(* PLC project batch, Dassault Systèmes ControlBuild 2020 *)
(* stored: creationDateTime 2019-04-23T11:14:51-01:00 *)

CONFIGURATION batch
  VAR_GLOBAL
    generalPanel/acknowledgePB AT 12 : BOOL := false;
    generalPanel/powerUp AT 6 : BOOL := false;
    generalPanel/emergencyStop AT 7 : BOOL := false;
    generalPanel/manualSwitch AT 8 : BOOL := false;
    generalPanel/autoSwitch AT 9 : BOOL := false;
    generalPanel/startCyclePB AT 10 : BOOL := false;
    generalPanel/endCyclePB AT 11 : BOOL := false;
    generalPanel/acknowledgePB/PB AT 12 : BOOL := false;
    generalPanel/acknowledgePB/action AT 26 : BOOL := false;
    generalPanel/acknowledgePB/timeCounter AT 17 : REAL := 0.0;
    generalPanel/acknowledgePB/pulseDuration AT 18 : REAL := 5.0;
    generalPanel/acknowledgePB/PBLogic AT 27 : BOOL := true;
    generalPanel/powerUp/PB AT 6 : BOOL := false;
    generalPanel/powerUp/action AT 28 : BOOL := false;
    generalPanel/powerUp/timeCounter AT 19 : REAL := 0.0;
    generalPanel/powerUp/pulseDuration AT 20 : REAL := 5.0;
    generalPanel/powerUp/PBLogic AT 29 : BOOL := true;
    generalPanel/modeSwitch/leftVariable AT 9 : BOOL := true;
    generalPanel/modeSwitch/rightVariable AT 8 : BOOL := false;
    generalPanel/modeSwitch/leftPosition AT 30 : BOOL := false;
    generalPanel/modeSwitch/rightPosition AT 31 : BOOL := false;
    generalPanel/startCyclePB/PB AT 10 : BOOL := false;
    generalPanel/startCyclePB/action AT 32 : BOOL := false;
    generalPanel/startCyclePB/timeCounter AT 21 : REAL := 0.0;
    generalPanel/startCyclePB/pulseDuration AT 22 : REAL := 5.0;
    generalPanel/startCyclePB/PBLogic AT 33 : BOOL := true;
    generalPanel/endCyclePB/PB AT 11 : BOOL := false;
    generalPanel/endCyclePB/action AT 34 : BOOL := false;
    generalPanel/endCyclePB/timeCounter AT 23 : REAL := 0.0;
    generalPanel/endCyclePB/pulseDuration AT 24 : REAL := 5.0;
    generalPanel/endCyclePB/PBLogic AT 35 : BOOL := true;
    generalPanel/bpCloture/PB AT 25 : BOOL := false;
    generalPanel/bpCloture/action AT 36 : BOOL := false;
    generalPanel/bpCloture/timeCounter AT 25 : REAL := 0.0;
    generalPanel/bpCloture/pulseDuration AT 26 : REAL := 5.0;
    generalPanel/bpCloture/PBLogic AT 37 : BOOL := true;
    generalPanel/emergencyStop/pb AT 7 : BOOL := false;
    generalPanel/emergencyStop/action AT 38 : BOOL := false;
    generalPanel/emergencyStop/PBLogic AT 39 : BOOL := false;
    recipe/flourWeight AT 523 : DINT := 0;
    recipe/syrup1Weight AT 524 : DINT := 0;
    recipe/syrup2Weight AT 525 : DINT := 0;
    recipe/syrup3Weight AT 526 : DINT := 0;
    recipe/recipeNumber AT 527 : DINT := 1;
    workingModes/powerUp AT 6 : BOOL := false;
    workingModes/emergencyStop AT 7 : BOOL := false;
    workingModes/manualSwitch AT 8 : BOOL := false;
    workingModes/autoSwitch AT 9 : BOOL := false;
    workingModes/startCyclePB AT 10 : BOOL := false;
    workingModes/endCyclePB AT 11 : BOOL := false;
    workingModes/acknowledgePB AT 12 : BOOL := false;
    workingModes/cycleEnd AT 13 : BOOL := false;
    workingModes/generalFault AT 14 : BOOL := false;
    workingModes/live AT 5 : BOOL := false;
    workingModes/autoMode AT 23 : BOOL := false;
    workingModes/manualMode AT 24 : BOOL := false;
    workingModes/cycleInProgress AT 15 : BOOL := false;
    workingModes/endCycleRequest AT 16 : BOOL := false;
    workingModes/emergencyStopState AT 40 : BOOL := false;
    management/cycleInProgress AT 15 : BOOL := false;
    management/endCycleRequest AT 16 : BOOL := false;
    management/kneadingOk AT 17 : BOOL := false;
    management/syrupWeighingOk AT 18 : BOOL := false;
    management/flourWeighingOk AT 19 : BOOL := false;
    management/cycleEnd AT 13 : BOOL := false;
    management/flourWeighingRq AT 20 : BOOL := false;
    management/syrupWeighingRq AT 21 : BOOL := false;
    management/kneadingRq AT 22 : BOOL := false;
    management/_X_10 AT 44 : BOOL := true;
    management/_X_11 AT 45 : BOOL := false;
    management/_X_12 AT 46 : BOOL := false;
    management/_X_13 AT 47 : BOOL := false;
    management/_X_14 AT 48 : BOOL := false;
    manufacturing/cycleInProgress AT 15 : BOOL := false;
    manufacturing/acknowledgePB AT 12 : BOOL := false;
    manufacturing/flourWeighingRequest AT 20 : BOOL := false;
    manufacturing/syrupWeighingRequest AT 21 : BOOL := false;
    manufacturing/kneadingRequest AT 22 : BOOL := false;
    manufacturing/autoMode AT 23 : BOOL := false;
    manufacturing/manualMode AT 24 : BOOL := false;
    manufacturing/flourWeight AT 523 : DINT := 0;
    manufacturing/syrup1Weight AT 524 : DINT := 0;
    manufacturing/syrup2Weight AT 525 : DINT := 0;
    manufacturing/syrup3Weight AT 526 : DINT := 0;
    manufacturing/generalFault AT 14 : BOOL := false;
    manufacturing/kneadingOK AT 17 : BOOL := false;
    manufacturing/flourWeighingOk AT 19 : BOOL := false;
    manufacturing/syrupWeighingOk AT 18 : BOOL := false;
    manufacturing/flour/cycleInProgress AT 15 : BOOL := false;
    manufacturing/flour/acknowledgePB AT 12 : BOOL := false;
    manufacturing/flour/weighingRequest AT 20 : BOOL := false;
    manufacturing/flour/flourWeight AT 523 : DINT := 0;
    manufacturing/flour/autoMode AT 23 : BOOL := false;
    manufacturing/flour/manualMode AT 24 : BOOL := false;
    manufacturing/flour/flourExtraction AT 28 : REAL := 0.0;
    manufacturing/flour/weighingOk AT 19 : BOOL := false;
    manufacturing/flour/fault AT 53 : BOOL := false;
    manufacturing/flour/airArrival/acknowledgePB AT 12 : BOOL := false;
    manufacturing/flour/airArrival/autoMode AT 23 : BOOL := false;
    manufacturing/flour/airArrival/manualMode AT 24 : BOOL := false;
    manufacturing/flour/airArrival/autoCloseCmd AT 62 : BOOL := false;
    manufacturing/flour/airArrival/autoOpenCmd AT 63 : BOOL := false;
    manufacturing/flour/airArrival/inputFlow AT 37 : REAL := 50.0;
    manufacturing/flour/airArrival/openedSensor AT 61 : BOOL := false;
    manufacturing/flour/airArrival/closedSensor AT 60 : BOOL := false;
    manufacturing/flour/airArrival/generalFault AT 66 : BOOL := false;
    manufacturing/flour/airArrival/outputFlow AT 39 : REAL := 0.0;
    manufacturing/flour/airArrival/percentOpening AT 36 : REAL := 0.0;
    manufacturing/flour/airArrival/panel1/closeValvePB AT 72 : BOOL := false;
    manufacturing/flour/airArrival/panel1/openValvePB AT 73 : BOOL := false;
    manufacturing/flour/airArrival/panel1/switch/leftVariable AT 72 : BOOL := false;
    manufacturing/flour/airArrival/panel1/switch/rightVariable AT 73 : BOOL := false;
    manufacturing/flour/airArrival/panel1/switch/leftPosition AT 76 : BOOL := false;
    manufacturing/flour/airArrival/panel1/switch/middlePosition AT 77 : BOOL := false;
    manufacturing/flour/airArrival/panel1/switch/rightPosition AT 78 : BOOL := false;
    manufacturing/flour/airArrival/cmdOfValve/autoMode AT 23 : BOOL := false;
    manufacturing/flour/airArrival/cmdOfValve/manualMode AT 24 : BOOL := false;
    manufacturing/flour/airArrival/cmdOfValve/closedSensorFB AT 60 : BOOL := false;
    manufacturing/flour/airArrival/cmdOfValve/openedSensorFB AT 61 : BOOL := false;
    manufacturing/flour/airArrival/cmdOfValve/autoCloseCmd AT 62 : BOOL := false;
    manufacturing/flour/airArrival/cmdOfValve/autoOpenCmd AT 63 : BOOL := false;
    manufacturing/flour/airArrival/cmdOfValve/closeValvePB AT 72 : BOOL := false;
    manufacturing/flour/airArrival/cmdOfValve/openValvePB AT 73 : BOOL := false;
    manufacturing/flour/airArrival/cmdOfValve/acknowledgePB AT 12 : BOOL := false;
    manufacturing/flour/airArrival/cmdOfValve/closeCmd AT 75 : BOOL := false;
    manufacturing/flour/airArrival/cmdOfValve/openCmd AT 74 : BOOL := false;
    manufacturing/flour/airArrival/cmdOfValve/generalFault AT 66 : BOOL := false;
    manufacturing/flour/airArrival/cmdOfValve/actions/autoMode AT 23 : BOOL := false;
    manufacturing/flour/airArrival/cmdOfValve/actions/manualMode AT 24 : BOOL := false;
    manufacturing/flour/airArrival/cmdOfValve/actions/autoCloseCmd AT 62 : BOOL := false;
    manufacturing/flour/airArrival/cmdOfValve/actions/autoOpenCmd AT 63 : BOOL := false;
    manufacturing/flour/airArrival/cmdOfValve/actions/closedSensorFB AT 60 : BOOL := false;
    manufacturing/flour/airArrival/cmdOfValve/actions/openedSensorFB AT 61 : BOOL := false;
    manufacturing/flour/airArrival/cmdOfValve/actions/closeValvePB AT 72 : BOOL := false;
    manufacturing/flour/airArrival/cmdOfValve/actions/openValvePB AT 73 : BOOL := false;
    manufacturing/flour/airArrival/cmdOfValve/actions/generalFault AT 66 : BOOL := false;
    manufacturing/flour/airArrival/cmdOfValve/actions/closeCmd AT 75 : BOOL := false;
    manufacturing/flour/airArrival/cmdOfValve/actions/openCmd AT 74 : BOOL := false;
    manufacturing/flour/airArrival/cmdOfValve/faults1/closeCmd AT 75 : BOOL := false;
    manufacturing/flour/airArrival/cmdOfValve/faults1/openCmd AT 74 : BOOL := false;
    manufacturing/flour/airArrival/cmdOfValve/faults1/closedSensorFB AT 60 : BOOL := false;
    manufacturing/flour/airArrival/cmdOfValve/faults1/openedSensorFB AT 61 : BOOL := false;
    manufacturing/flour/airArrival/cmdOfValve/faults1/acknowledgePB AT 12 : BOOL := false;
    manufacturing/flour/airArrival/cmdOfValve/faults1/generalFault AT 66 : BOOL := false;
    manufacturing/flour/airArrival/cmdOfValve/faults1/closedSensorFault AT 79 : BOOL := false;
    manufacturing/flour/airArrival/cmdOfValve/faults1/openedSensorFault AT 80 : BOOL := false;
    manufacturing/flour/airArrival/cmdOfValve/faults1/discordanceFault AT 81 : BOOL := false;
    manufacturing/flour/airArrival/cmdOfValve/faults1/presetMvt AT 542 : TIME := T#0h0m4s0ms;
    manufacturing/flour/airArrival/cmdOfValve/faults1/presetDiscordance AT 546 : TIME := T#0h0m0s200ms;
    manufacturing/flour/airArrival/valve/voltage380 AT 71 : BOOL := true;
    manufacturing/flour/airArrival/valve/cmdSupply AT 70 : BOOL := true;
    manufacturing/flour/airArrival/valve/sensorSupply AT 69 : BOOL := true;
    manufacturing/flour/airArrival/valve/openCmd AT 74 : BOOL := false;
    manufacturing/flour/airArrival/valve/closeCmd AT 75 : BOOL := false;
    manufacturing/flour/airArrival/valve/inputFlow AT 37 : REAL := 50.0;
    manufacturing/flour/airArrival/valve/openedSensor AT 61 : BOOL := false;
    manufacturing/flour/airArrival/valve/closedSensor AT 60 : BOOL := false;
    manufacturing/flour/airArrival/valve/outputFlow AT 39 : REAL := 0.0;
    manufacturing/flour/airArrival/valve/percentOpening AT 36 : REAL := 0.0;
    manufacturing/flour/airArrival/valve/increment AT 45 : REAL := 0.0;
    manufacturing/flour/airArrival/valve/memoOpen AT 91 : BOOL := false;
    manufacturing/flour/airArrival/valve/memoClose AT 92 : BOOL := false;
    manufacturing/flour/airArrival/valve/openState AT 93 : BOOL := false;
    manufacturing/flour/airArrival/valve/closeState AT 94 : BOOL := false;
    manufacturing/flour/airArrival/valve/openingVal AT 46 : REAL := 0.0;
    manufacturing/flour/airArrival/valve/unit AT 47 : REAL := 0.0;
    manufacturing/flour/airArrival/valve/openingTime AT 48 : REAL := 0.5;
    manufacturing/flour/airArrival/valve/openedSensorLogic AT 95 : BOOL := true;
    manufacturing/flour/airArrival/valve/closedSensorLogic AT 96 : BOOL := true;
    manufacturing/flour/airArrival/valve/flowMax AT 49 : REAL := 10000.0;
    manufacturing/flour/airArrival/valve/flowPerHour AT 97 : BOOL := true;
    manufacturing/flour/airArrival/valve/flowPerMinute AT 98 : BOOL := false;
    manufacturing/flour/airArrival/valve/d_locking AT 99 : BOOL := false;
    manufacturing/flour/airArrival/valve/v_d_locking AT 50 : REAL := 2.0;
    manufacturing/flour/airArrival/valve/d_flow AT 100 : BOOL := false;
    manufacturing/flour/airArrival/valve/v_d_flow AT 51 : REAL := 2.0;
    manufacturing/flour/airArrival/valve/d_electrical AT 101 : BOOL := false;
    manufacturing/flour/airArrival/valve/v_d_electrical AT 102 : BOOL := false;
    manufacturing/flour/airArrival/valve/d_closedSensor AT 103 : BOOL := false;
    manufacturing/flour/airArrival/valve/v_d_closedSensor AT 104 : BOOL := false;
    manufacturing/flour/airArrival/valve/d_openedSensor AT 105 : BOOL := false;
    manufacturing/flour/airArrival/valve/v_d_openedSensor AT 106 : BOOL := false;
    manufacturing/flour/extractingValve/acknowledgePB AT 12 : BOOL := false;
    manufacturing/flour/extractingValve/autoMode AT 23 : BOOL := false;
    manufacturing/flour/extractingValve/manualMode AT 24 : BOOL := false;
    manufacturing/flour/extractingValve/autoCloseCmd AT 64 : BOOL := false;
    manufacturing/flour/extractingValve/autoOpenCmd AT 65 : BOOL := false;
    manufacturing/flour/extractingValve/inputFlow AT 38 : REAL := 0.0;
    manufacturing/flour/extractingValve/openedSensor AT 59 : BOOL := false;
    manufacturing/flour/extractingValve/closedSensor AT 58 : BOOL := false;
    manufacturing/flour/extractingValve/generalFault AT 68 : BOOL := false;
    manufacturing/flour/extractingValve/outputFlow AT 28 : REAL := 0.0;
    manufacturing/flour/extractingValve/percentOpening AT 35 : REAL := 0.0;
    manufacturing/flour/extractingValve/panel1/closeValvePB AT 110 : BOOL := false;
    manufacturing/flour/extractingValve/panel1/openValvePB AT 111 : BOOL := false;
    manufacturing/flour/extractingValve/panel1/switch/leftVariable AT 110 : BOOL := false;
    manufacturing/flour/extractingValve/panel1/switch/rightVariable AT 111 : BOOL := false;
    manufacturing/flour/extractingValve/panel1/switch/leftPosition AT 114 : BOOL := false;
    manufacturing/flour/extractingValve/panel1/switch/middlePosition AT 115 : BOOL := false;
    manufacturing/flour/extractingValve/panel1/switch/rightPosition AT 116 : BOOL := false;
    manufacturing/flour/extractingValve/cmdOfValve/autoMode AT 23 : BOOL := false;
    manufacturing/flour/extractingValve/cmdOfValve/manualMode AT 24 : BOOL := false;
    manufacturing/flour/extractingValve/cmdOfValve/closedSensorFB AT 58 : BOOL := false;
    manufacturing/flour/extractingValve/cmdOfValve/openedSensorFB AT 59 : BOOL := false;
    manufacturing/flour/extractingValve/cmdOfValve/autoCloseCmd AT 64 : BOOL := false;
    manufacturing/flour/extractingValve/cmdOfValve/autoOpenCmd AT 65 : BOOL := false;
    manufacturing/flour/extractingValve/cmdOfValve/closeValvePB AT 110 : BOOL := false;
    manufacturing/flour/extractingValve/cmdOfValve/openValvePB AT 111 : BOOL := false;
    manufacturing/flour/extractingValve/cmdOfValve/acknowledgePB AT 12 : BOOL := false;
    manufacturing/flour/extractingValve/cmdOfValve/closeCmd AT 113 : BOOL := false;
    manufacturing/flour/extractingValve/cmdOfValve/openCmd AT 112 : BOOL := false;
    manufacturing/flour/extractingValve/cmdOfValve/generalFault AT 68 : BOOL := false;
    manufacturing/flour/extractingValve/cmdOfValve/actions/autoMode AT 23 : BOOL := false;
    manufacturing/flour/extractingValve/cmdOfValve/actions/manualMode AT 24 : BOOL := false;
    manufacturing/flour/extractingValve/cmdOfValve/actions/autoCloseCmd AT 64 : BOOL := false;
    manufacturing/flour/extractingValve/cmdOfValve/actions/autoOpenCmd AT 65 : BOOL := false;
    manufacturing/flour/extractingValve/cmdOfValve/actions/closedSensorFB AT 58 : BOOL := false;
    manufacturing/flour/extractingValve/cmdOfValve/actions/openedSensorFB AT 59 : BOOL := false;
    manufacturing/flour/extractingValve/cmdOfValve/actions/closeValvePB AT 110 : BOOL := false;
    manufacturing/flour/extractingValve/cmdOfValve/actions/openValvePB AT 111 : BOOL := false;
    manufacturing/flour/extractingValve/cmdOfValve/actions/generalFault AT 68 : BOOL := false;
    manufacturing/flour/extractingValve/cmdOfValve/actions/closeCmd AT 113 : BOOL := false;
    manufacturing/flour/extractingValve/cmdOfValve/actions/openCmd AT 112 : BOOL := false;
    manufacturing/flour/extractingValve/cmdOfValve/faults1/closeCmd AT 113 : BOOL := false;
    manufacturing/flour/extractingValve/cmdOfValve/faults1/openCmd AT 112 : BOOL := false;
    manufacturing/flour/extractingValve/cmdOfValve/faults1/closedSensorFB AT 58 : BOOL := false;
    manufacturing/flour/extractingValve/cmdOfValve/faults1/openedSensorFB AT 59 : BOOL := false;
    manufacturing/flour/extractingValve/cmdOfValve/faults1/acknowledgePB AT 12 : BOOL := false;
    manufacturing/flour/extractingValve/cmdOfValve/faults1/generalFault AT 68 : BOOL := false;
    manufacturing/flour/extractingValve/cmdOfValve/faults1/closedSensorFault AT 117 : BOOL := false;
    manufacturing/flour/extractingValve/cmdOfValve/faults1/openedSensorFault AT 118 : BOOL := false;
    manufacturing/flour/extractingValve/cmdOfValve/faults1/discordanceFault AT 119 : BOOL := false;
    manufacturing/flour/extractingValve/cmdOfValve/faults1/presetMvt AT 583 : TIME := T#0h0m4s0ms;
    manufacturing/flour/extractingValve/cmdOfValve/faults1/presetDiscordance AT 587 : TIME := T#0h0m0s200ms;
    manufacturing/flour/extractingValve/valve/voltage380 AT 109 : BOOL := true;
    manufacturing/flour/extractingValve/valve/cmdSupply AT 108 : BOOL := true;
    manufacturing/flour/extractingValve/valve/sensorSupply AT 107 : BOOL := true;
    manufacturing/flour/extractingValve/valve/openCmd AT 112 : BOOL := false;
    manufacturing/flour/extractingValve/valve/closeCmd AT 113 : BOOL := false;
    manufacturing/flour/extractingValve/valve/inputFlow AT 38 : REAL := 0.0;
    manufacturing/flour/extractingValve/valve/openedSensor AT 59 : BOOL := false;
    manufacturing/flour/extractingValve/valve/closedSensor AT 58 : BOOL := false;
    manufacturing/flour/extractingValve/valve/outputFlow AT 28 : REAL := 0.0;
    manufacturing/flour/extractingValve/valve/percentOpening AT 35 : REAL := 0.0;
    manufacturing/flour/extractingValve/valve/increment AT 55 : REAL := 0.0;
    manufacturing/flour/extractingValve/valve/memoOpen AT 129 : BOOL := false;
    manufacturing/flour/extractingValve/valve/memoClose AT 130 : BOOL := false;
    manufacturing/flour/extractingValve/valve/openState AT 131 : BOOL := false;
    manufacturing/flour/extractingValve/valve/closeState AT 132 : BOOL := false;
    manufacturing/flour/extractingValve/valve/openingVal AT 56 : REAL := 0.0;
    manufacturing/flour/extractingValve/valve/unit AT 57 : REAL := 0.0;
    manufacturing/flour/extractingValve/valve/openingTime AT 58 : REAL := 0.5;
    manufacturing/flour/extractingValve/valve/openedSensorLogic AT 133 : BOOL := true;
    manufacturing/flour/extractingValve/valve/closedSensorLogic AT 134 : BOOL := true;
    manufacturing/flour/extractingValve/valve/flowMax AT 59 : REAL := 10000.0;
    manufacturing/flour/extractingValve/valve/flowPerHour AT 135 : BOOL := true;
    manufacturing/flour/extractingValve/valve/flowPerMinute AT 136 : BOOL := false;
    manufacturing/flour/extractingValve/valve/d_locking AT 137 : BOOL := false;
    manufacturing/flour/extractingValve/valve/v_d_locking AT 60 : REAL := 2.0;
    manufacturing/flour/extractingValve/valve/d_flow AT 138 : BOOL := false;
    manufacturing/flour/extractingValve/valve/v_d_flow AT 61 : REAL := 2.0;
    manufacturing/flour/extractingValve/valve/d_electrical AT 139 : BOOL := false;
    manufacturing/flour/extractingValve/valve/v_d_electrical AT 140 : BOOL := false;
    manufacturing/flour/extractingValve/valve/d_closedSensor AT 141 : BOOL := false;
    manufacturing/flour/extractingValve/valve/v_d_closedSensor AT 142 : BOOL := false;
    manufacturing/flour/extractingValve/valve/d_openedSensor AT 143 : BOOL := false;
    manufacturing/flour/extractingValve/valve/v_d_openedSensor AT 144 : BOOL := false;
    manufacturing/flour/airExtraction/acknowledgePB AT 12 : BOOL := false;
    manufacturing/flour/airExtraction/autoMode AT 23 : BOOL := false;
    manufacturing/flour/airExtraction/manualMode AT 24 : BOOL := false;
    manufacturing/flour/airExtraction/autoCloseCmd AT 64 : BOOL := false;
    manufacturing/flour/airExtraction/autoOpenCmd AT 65 : BOOL := false;
    manufacturing/flour/airExtraction/inputFlow AT 34 : REAL := 0.0;
    manufacturing/flour/airExtraction/openedSensor AT 57 : BOOL := false;
    manufacturing/flour/airExtraction/closedSensor AT 56 : BOOL := false;
    manufacturing/flour/airExtraction/generalFault AT 67 : BOOL := false;
    manufacturing/flour/airExtraction/outputFlow AT 33 : REAL := 0.0;
    manufacturing/flour/airExtraction/percentOpening AT 32 : REAL := 0.0;
    manufacturing/flour/airExtraction/panel1/closeValvePB AT 148 : BOOL := false;
    manufacturing/flour/airExtraction/panel1/openValvePB AT 149 : BOOL := false;
    manufacturing/flour/airExtraction/panel1/switch/leftVariable AT 148 : BOOL := false;
    manufacturing/flour/airExtraction/panel1/switch/rightVariable AT 149 : BOOL := false;
    manufacturing/flour/airExtraction/panel1/switch/leftPosition AT 152 : BOOL := false;
    manufacturing/flour/airExtraction/panel1/switch/middlePosition AT 153 : BOOL := false;
    manufacturing/flour/airExtraction/panel1/switch/rightPosition AT 154 : BOOL := false;
    manufacturing/flour/airExtraction/cmdOfValve/autoMode AT 23 : BOOL := false;
    manufacturing/flour/airExtraction/cmdOfValve/manualMode AT 24 : BOOL := false;
    manufacturing/flour/airExtraction/cmdOfValve/closedSensorFB AT 56 : BOOL := false;
    manufacturing/flour/airExtraction/cmdOfValve/openedSensorFB AT 57 : BOOL := false;
    manufacturing/flour/airExtraction/cmdOfValve/autoCloseCmd AT 64 : BOOL := false;
    manufacturing/flour/airExtraction/cmdOfValve/autoOpenCmd AT 65 : BOOL := false;
    manufacturing/flour/airExtraction/cmdOfValve/closeValvePB AT 148 : BOOL := false;
    manufacturing/flour/airExtraction/cmdOfValve/openValvePB AT 149 : BOOL := false;
    manufacturing/flour/airExtraction/cmdOfValve/acknowledgePB AT 12 : BOOL := false;
    manufacturing/flour/airExtraction/cmdOfValve/closeCmd AT 151 : BOOL := false;
    manufacturing/flour/airExtraction/cmdOfValve/openCmd AT 150 : BOOL := false;
    manufacturing/flour/airExtraction/cmdOfValve/generalFault AT 67 : BOOL := false;
    manufacturing/flour/airExtraction/cmdOfValve/actions/autoMode AT 23 : BOOL := false;
    manufacturing/flour/airExtraction/cmdOfValve/actions/manualMode AT 24 : BOOL := false;
    manufacturing/flour/airExtraction/cmdOfValve/actions/autoCloseCmd AT 64 : BOOL := false;
    manufacturing/flour/airExtraction/cmdOfValve/actions/autoOpenCmd AT 65 : BOOL := false;
    manufacturing/flour/airExtraction/cmdOfValve/actions/closedSensorFB AT 56 : BOOL := false;
    manufacturing/flour/airExtraction/cmdOfValve/actions/openedSensorFB AT 57 : BOOL := false;
    manufacturing/flour/airExtraction/cmdOfValve/actions/closeValvePB AT 148 : BOOL := false;
    manufacturing/flour/airExtraction/cmdOfValve/actions/openValvePB AT 149 : BOOL := false;
    manufacturing/flour/airExtraction/cmdOfValve/actions/generalFault AT 67 : BOOL := false;
    manufacturing/flour/airExtraction/cmdOfValve/actions/closeCmd AT 151 : BOOL := false;
    manufacturing/flour/airExtraction/cmdOfValve/actions/openCmd AT 150 : BOOL := false;
    manufacturing/flour/airExtraction/cmdOfValve/faults1/closeCmd AT 151 : BOOL := false;
    manufacturing/flour/airExtraction/cmdOfValve/faults1/openCmd AT 150 : BOOL := false;
    manufacturing/flour/airExtraction/cmdOfValve/faults1/closedSensorFB AT 56 : BOOL := false;
    manufacturing/flour/airExtraction/cmdOfValve/faults1/openedSensorFB AT 57 : BOOL := false;
    manufacturing/flour/airExtraction/cmdOfValve/faults1/acknowledgePB AT 12 : BOOL := false;
    manufacturing/flour/airExtraction/cmdOfValve/faults1/generalFault AT 67 : BOOL := false;
    manufacturing/flour/airExtraction/cmdOfValve/faults1/closedSensorFault AT 155 : BOOL := false;
    manufacturing/flour/airExtraction/cmdOfValve/faults1/openedSensorFault AT 156 : BOOL := false;
    manufacturing/flour/airExtraction/cmdOfValve/faults1/discordanceFault AT 157 : BOOL := false;
    manufacturing/flour/airExtraction/cmdOfValve/faults1/presetMvt AT 624 : TIME := T#0h0m4s0ms;
    manufacturing/flour/airExtraction/cmdOfValve/faults1/presetDiscordance AT 628 : TIME := T#0h0m0s200ms;
    manufacturing/flour/airExtraction/valve/voltage380 AT 147 : BOOL := true;
    manufacturing/flour/airExtraction/valve/cmdSupply AT 146 : BOOL := true;
    manufacturing/flour/airExtraction/valve/sensorSupply AT 145 : BOOL := true;
    manufacturing/flour/airExtraction/valve/openCmd AT 150 : BOOL := false;
    manufacturing/flour/airExtraction/valve/closeCmd AT 151 : BOOL := false;
    manufacturing/flour/airExtraction/valve/inputFlow AT 34 : REAL := 0.0;
    manufacturing/flour/airExtraction/valve/openedSensor AT 57 : BOOL := false;
    manufacturing/flour/airExtraction/valve/closedSensor AT 56 : BOOL := false;
    manufacturing/flour/airExtraction/valve/outputFlow AT 33 : REAL := 0.0;
    manufacturing/flour/airExtraction/valve/percentOpening AT 32 : REAL := 0.0;
    manufacturing/flour/airExtraction/valve/increment AT 65 : REAL := 0.0;
    manufacturing/flour/airExtraction/valve/memoOpen AT 167 : BOOL := false;
    manufacturing/flour/airExtraction/valve/memoClose AT 168 : BOOL := false;
    manufacturing/flour/airExtraction/valve/openState AT 169 : BOOL := false;
    manufacturing/flour/airExtraction/valve/closeState AT 170 : BOOL := false;
    manufacturing/flour/airExtraction/valve/openingVal AT 66 : REAL := 0.0;
    manufacturing/flour/airExtraction/valve/unit AT 67 : REAL := 0.0;
    manufacturing/flour/airExtraction/valve/openingTime AT 68 : REAL := 0.5;
    manufacturing/flour/airExtraction/valve/openedSensorLogic AT 171 : BOOL := true;
    manufacturing/flour/airExtraction/valve/closedSensorLogic AT 172 : BOOL := true;
    manufacturing/flour/airExtraction/valve/flowMax AT 69 : REAL := 10000.0;
    manufacturing/flour/airExtraction/valve/flowPerHour AT 173 : BOOL := true;
    manufacturing/flour/airExtraction/valve/flowPerMinute AT 174 : BOOL := false;
    manufacturing/flour/airExtraction/valve/d_locking AT 175 : BOOL := false;
    manufacturing/flour/airExtraction/valve/v_d_locking AT 70 : REAL := 2.0;
    manufacturing/flour/airExtraction/valve/d_flow AT 176 : BOOL := false;
    manufacturing/flour/airExtraction/valve/v_d_flow AT 71 : REAL := 2.0;
    manufacturing/flour/airExtraction/valve/d_electrical AT 177 : BOOL := false;
    manufacturing/flour/airExtraction/valve/v_d_electrical AT 178 : BOOL := false;
    manufacturing/flour/airExtraction/valve/d_closedSensor AT 179 : BOOL := false;
    manufacturing/flour/airExtraction/valve/v_d_closedSensor AT 180 : BOOL := false;
    manufacturing/flour/airExtraction/valve/d_openedSensor AT 181 : BOOL := false;
    manufacturing/flour/airExtraction/valve/v_d_openedSensor AT 182 : BOOL := false;
    manufacturing/flour/flourWeighing/inletFlow AT 39 : REAL := 0.0;
    manufacturing/flour/flourWeighing/outletFlow AT 28 : REAL := 0.0;
    manufacturing/flour/flourWeighing/tankLevel AT 40 : REAL := 0.0;
    manufacturing/flour/flourWeighing/percent AT 72 : REAL := 0.0;
    manufacturing/flour/flourWeighing/capacity AT 73 : REAL := 100.0;
    manufacturing/flour/flourWeighing/d_level AT 183 : BOOL := false;
    manufacturing/flour/flourWeighing/v_d_level AT 74 : REAL := 0.0;
    manufacturing/flour/flow/inputFlow AT 40 : REAL := 0.0;
    manufacturing/flour/flow/outputFlow AT 38 : REAL := 0.0;
    manufacturing/flour/flow/unit AT 75 : REAL := 0.0;
    manufacturing/flour/flow/flowMax AT 76 : REAL := 20000.0;
    manufacturing/flour/flow/flowPerHour AT 184 : BOOL := true;
    manufacturing/flour/flow/flowPerMinute AT 185 : BOOL := false;
    manufacturing/flour/level/measure AT 40 : REAL := 0.0;
    manufacturing/flour/level/sensorSupply AT 55 : BOOL := true;
    manufacturing/flour/level/realValue AT 41 : REAL := 0.0;
    manufacturing/flour/level/intValue AT 31 : REAL := 0.0;
    manufacturing/flour/level/dintValue AT 30 : REAL := 0.0;
    manufacturing/flour/level/tmp AT 656 : DINT := 0;
    manufacturing/flour/level/localValue AT 77 : REAL := 0.0;
    manufacturing/flour/level/nbDigit AT 657 : SINT := 2;
    manufacturing/flour/level/d_value AT 186 : BOOL := false;
    manufacturing/flour/level/v_d_value AT 78 : REAL := 0.0;
    manufacturing/flour/faults1/generalFault3 AT 66 : BOOL := false;
    manufacturing/flour/faults1/generalFault2 AT 67 : BOOL := false;
    manufacturing/flour/faults1/generalFault1 AT 68 : BOOL := false;
    manufacturing/flour/faults1/fault AT 53 : BOOL := false;
    manufacturing/flour/flourManagement/weighingRequest AT 20 : BOOL := false;
    manufacturing/flour/flourManagement/cycleInProgress AT 15 : BOOL := false;
    manufacturing/flour/flourManagement/weighedWeight AT 532 : DINT := 0;
    manufacturing/flour/flourManagement/flourWeight AT 523 : DINT := 0;
    manufacturing/flour/flourManagement/weighingOk AT 19 : BOOL := false;
    manufacturing/flour/flourManagement/introduceFlour AT 63 : BOOL := false;
    manufacturing/flour/flourManagement/introFlourEnd AT 62 : BOOL := false;
    manufacturing/flour/flourManagement/exitFlour AT 65 : BOOL := false;
    manufacturing/flour/flourManagement/exitFlourEnd AT 64 : BOOL := false;
    manufacturing/flour/flourManagement/totalWeight AT 658 : DINT := 0;
    manufacturing/flour/flourManagement/endOfWeighing AT 187 : BOOL := false;
    manufacturing/flour/flourManagement/_X_10 AT 188 : BOOL := true;
    manufacturing/flour/flourManagement/_X_11 AT 189 : BOOL := false;
    manufacturing/flour/flourManagement/_X_12 AT 190 : BOOL := false;
    manufacturing/flour/flourManagement/_X_13 AT 191 : BOOL := false;
    manufacturing/flour/flourManagement/_X_14 AT 192 : BOOL := false;
    manufacturing/flour/flourManagement/_X_15 AT 193 : BOOL := false;
    manufacturing/flour/flourManagement/maxWeight AT 659 : DINT := 100;
    manufacturing/flour/scale/inputValue AT 41 : REAL := 0.0;
    manufacturing/flour/scale/realValue AT 29 : REAL := 0.0;
    manufacturing/flour/scale/dintValue AT 532 : DINT := 0;
    manufacturing/flour/scale/intValue AT 531 : INT := 0;
    manufacturing/flour/scale/a AT 79 : REAL := 0.0;
    manufacturing/flour/scale/b AT 80 : REAL := 0.0;
    manufacturing/flour/scale/k AT 81 : REAL := 0.0;
    manufacturing/flour/scale/minInput AT 82 : REAL := 0.0;
    manufacturing/flour/scale/maxInput AT 83 : REAL := 100.0;
    manufacturing/flour/scale/minOutput AT 84 : REAL := 0.0;
    manufacturing/flour/scale/maxOutput AT 85 : REAL := 100.0;
    manufacturing/flour/scale/d_scale AT 198 : BOOL := false;
    manufacturing/flour/scale/v_d_scale AT 86 : REAL := 0.0;
    manufacturing/syrup/syrup1Weight AT 524 : DINT := 0;
    manufacturing/syrup/syrup2Weight AT 525 : DINT := 0;
    manufacturing/syrup/syrup3Weight AT 526 : DINT := 0;
    manufacturing/syrup/cycleInProgress AT 15 : BOOL := false;
    manufacturing/syrup/weighingRequest AT 21 : BOOL := false;
    manufacturing/syrup/acknowledgePB AT 12 : BOOL := false;
    manufacturing/syrup/autoMode AT 23 : BOOL := false;
    manufacturing/syrup/manualMode AT 24 : BOOL := false;
    manufacturing/syrup/weighingOk AT 18 : BOOL := false;
    manufacturing/syrup/fault AT 54 : BOOL := false;
    manufacturing/syrup/syrupExtraction AT 27 : REAL := 0.0;
    manufacturing/syrup/flow/inputFlow AT 97 : REAL := 0.0;
    manufacturing/syrup/flow/outputFlow AT 98 : REAL := 0.0;
    manufacturing/syrup/flow/unit AT 104 : REAL := 0.0;
    manufacturing/syrup/flow/flowMax AT 105 : REAL := 40000.0;
    manufacturing/syrup/flow/flowPerHour AT 220 : BOOL := true;
    manufacturing/syrup/flow/flowPerMinute AT 221 : BOOL := false;
    manufacturing/syrup/syrupManagement/weighingRequest AT 21 : BOOL := false;
    manufacturing/syrup/syrupManagement/cycleInProgress AT 15 : BOOL := false;
    manufacturing/syrup/syrupManagement/weighingWeight AT 662 : DINT := 0;
    manufacturing/syrup/syrupManagement/syrup1Weight AT 524 : DINT := 0;
    manufacturing/syrup/syrupManagement/syrup2Weight AT 525 : DINT := 0;
    manufacturing/syrup/syrupManagement/syrup3Weight AT 526 : DINT := 0;
    manufacturing/syrup/syrupManagement/weighingOk AT 18 : BOOL := false;
    manufacturing/syrup/syrupManagement/introduceS1 AT 209 : BOOL := false;
    manufacturing/syrup/syrupManagement/introS1End AT 208 : BOOL := false;
    manufacturing/syrup/syrupManagement/introduceS2 AT 211 : BOOL := false;
    manufacturing/syrup/syrupManagement/introS2End AT 210 : BOOL := false;
    manufacturing/syrup/syrupManagement/introduceS3 AT 213 : BOOL := false;
    manufacturing/syrup/syrupManagement/introS3End AT 212 : BOOL := false;
    manufacturing/syrup/syrupManagement/exitSyrup AT 215 : BOOL := false;
    manufacturing/syrup/syrupManagement/exitSyrupEnd AT 214 : BOOL := false;
    manufacturing/syrup/syrupManagement/totalWeight AT 663 : DINT := 0;
    manufacturing/syrup/syrupManagement/weighingS1 AT 222 : BOOL := false;
    manufacturing/syrup/syrupManagement/weighingS2 AT 223 : BOOL := false;
    manufacturing/syrup/syrupManagement/weighingS3 AT 224 : BOOL := false;
    manufacturing/syrup/syrupManagement/weighingS1Ok AT 225 : BOOL := false;
    manufacturing/syrup/syrupManagement/weighingS2Ok AT 226 : BOOL := false;
    manufacturing/syrup/syrupManagement/weighingS3Ok AT 227 : BOOL := false;
    manufacturing/syrup/syrupManagement/endOfWeighingS3 AT 228 : BOOL := false;
    manufacturing/syrup/syrupManagement/endOfWeighingS2 AT 229 : BOOL := false;
    manufacturing/syrup/syrupManagement/endOfWeighingS1 AT 230 : BOOL := false;
    manufacturing/syrup/syrupManagement/_X_10 AT 231 : BOOL := true;
    manufacturing/syrup/syrupManagement/_X_11 AT 232 : BOOL := false;
    manufacturing/syrup/syrupManagement/_X_12 AT 233 : BOOL := false;
    manufacturing/syrup/syrupManagement/_X_13 AT 234 : BOOL := false;
    manufacturing/syrup/syrupManagement/_X_14 AT 235 : BOOL := false;
    manufacturing/syrup/syrupManagement/_X_15 AT 236 : BOOL := false;
    manufacturing/syrup/syrupManagement/_X_20 AT 237 : BOOL := true;
    manufacturing/syrup/syrupManagement/_X_21 AT 238 : BOOL := false;
    manufacturing/syrup/syrupManagement/_X_22 AT 239 : BOOL := false;
    manufacturing/syrup/syrupManagement/_X_23 AT 240 : BOOL := false;
    manufacturing/syrup/syrupManagement/_X_24 AT 241 : BOOL := false;
    manufacturing/syrup/syrupManagement/_X_30 AT 242 : BOOL := true;
    manufacturing/syrup/syrupManagement/_X_31 AT 243 : BOOL := false;
    manufacturing/syrup/syrupManagement/_X_32 AT 244 : BOOL := false;
    manufacturing/syrup/syrupManagement/_X_33 AT 247 : BOOL := false;
    manufacturing/syrup/syrupManagement/_X_34 AT 245 : BOOL := false;
    manufacturing/syrup/syrupManagement/_X_35 AT 246 : BOOL := false;
    manufacturing/syrup/syrupManagement/_X_40 AT 248 : BOOL := true;
    manufacturing/syrup/syrupManagement/_X_41 AT 249 : BOOL := false;
    manufacturing/syrup/syrupManagement/_X_42 AT 250 : BOOL := false;
    manufacturing/syrup/syrupManagement/_X_43 AT 253 : BOOL := false;
    manufacturing/syrup/syrupManagement/_X_44 AT 251 : BOOL := false;
    manufacturing/syrup/syrupManagement/_X_45 AT 252 : BOOL := false;
    manufacturing/syrup/syrupManagement/maxWeight AT 664 : DINT := 200;
    manufacturing/syrup/arrivalValveSyrup1/acknowledgePB AT 12 : BOOL := false;
    manufacturing/syrup/arrivalValveSyrup1/autoMode AT 23 : BOOL := false;
    manufacturing/syrup/arrivalValveSyrup1/manualMode AT 24 : BOOL := false;
    manufacturing/syrup/arrivalValveSyrup1/autoCloseCmd AT 208 : BOOL := false;
    manufacturing/syrup/arrivalValveSyrup1/autoOpenCmd AT 209 : BOOL := false;
    manufacturing/syrup/arrivalValveSyrup1/inputFlow AT 96 : REAL := 50.0;
    manufacturing/syrup/arrivalValveSyrup1/openedSensor AT 207 : BOOL := false;
    manufacturing/syrup/arrivalValveSyrup1/closedSensor AT 206 : BOOL := false;
    manufacturing/syrup/arrivalValveSyrup1/generalFault AT 216 : BOOL := false;
    manufacturing/syrup/arrivalValveSyrup1/outputFlow AT 99 : REAL := 0.0;
    manufacturing/syrup/arrivalValveSyrup1/percentOpening AT 95 : REAL := 0.0;
    manufacturing/syrup/arrivalValveSyrup1/panel1/closeValvePB AT 273 : BOOL := false;
    manufacturing/syrup/arrivalValveSyrup1/panel1/openValvePB AT 274 : BOOL := false;
    manufacturing/syrup/arrivalValveSyrup1/panel1/switch/leftVariable AT 273 : BOOL := false;
    manufacturing/syrup/arrivalValveSyrup1/panel1/switch/rightVariable AT 274 : BOOL := false;
    manufacturing/syrup/arrivalValveSyrup1/panel1/switch/leftPosition AT 277 : BOOL := false;
    manufacturing/syrup/arrivalValveSyrup1/panel1/switch/middlePosition AT 278 : BOOL := false;
    manufacturing/syrup/arrivalValveSyrup1/panel1/switch/rightPosition AT 279 : BOOL := false;
    manufacturing/syrup/arrivalValveSyrup1/cmdOfValve/autoMode AT 23 : BOOL := false;
    manufacturing/syrup/arrivalValveSyrup1/cmdOfValve/manualMode AT 24 : BOOL := false;
    manufacturing/syrup/arrivalValveSyrup1/cmdOfValve/closedSensorFB AT 206 : BOOL := false;
    manufacturing/syrup/arrivalValveSyrup1/cmdOfValve/openedSensorFB AT 207 : BOOL := false;
    manufacturing/syrup/arrivalValveSyrup1/cmdOfValve/autoCloseCmd AT 208 : BOOL := false;
    manufacturing/syrup/arrivalValveSyrup1/cmdOfValve/autoOpenCmd AT 209 : BOOL := false;
    manufacturing/syrup/arrivalValveSyrup1/cmdOfValve/closeValvePB AT 273 : BOOL := false;
    manufacturing/syrup/arrivalValveSyrup1/cmdOfValve/openValvePB AT 274 : BOOL := false;
    manufacturing/syrup/arrivalValveSyrup1/cmdOfValve/acknowledgePB AT 12 : BOOL := false;
    manufacturing/syrup/arrivalValveSyrup1/cmdOfValve/closeCmd AT 276 : BOOL := false;
    manufacturing/syrup/arrivalValveSyrup1/cmdOfValve/openCmd AT 275 : BOOL := false;
    manufacturing/syrup/arrivalValveSyrup1/cmdOfValve/generalFault AT 216 : BOOL := false;
    manufacturing/syrup/arrivalValveSyrup1/cmdOfValve/actions/autoMode AT 23 : BOOL := false;
    manufacturing/syrup/arrivalValveSyrup1/cmdOfValve/actions/manualMode AT 24 : BOOL := false;
    manufacturing/syrup/arrivalValveSyrup1/cmdOfValve/actions/autoCloseCmd AT 208 : BOOL := false;
    manufacturing/syrup/arrivalValveSyrup1/cmdOfValve/actions/autoOpenCmd AT 209 : BOOL := false;
    manufacturing/syrup/arrivalValveSyrup1/cmdOfValve/actions/closedSensorFB AT 206 : BOOL := false;
    manufacturing/syrup/arrivalValveSyrup1/cmdOfValve/actions/openedSensorFB AT 207 : BOOL := false;
    manufacturing/syrup/arrivalValveSyrup1/cmdOfValve/actions/closeValvePB AT 273 : BOOL := false;
    manufacturing/syrup/arrivalValveSyrup1/cmdOfValve/actions/openValvePB AT 274 : BOOL := false;
    manufacturing/syrup/arrivalValveSyrup1/cmdOfValve/actions/generalFault AT 216 : BOOL := false;
    manufacturing/syrup/arrivalValveSyrup1/cmdOfValve/actions/closeCmd AT 276 : BOOL := false;
    manufacturing/syrup/arrivalValveSyrup1/cmdOfValve/actions/openCmd AT 275 : BOOL := false;
    manufacturing/syrup/arrivalValveSyrup1/cmdOfValve/faults1/closeCmd AT 276 : BOOL := false;
    manufacturing/syrup/arrivalValveSyrup1/cmdOfValve/faults1/openCmd AT 275 : BOOL := false;
    manufacturing/syrup/arrivalValveSyrup1/cmdOfValve/faults1/closedSensorFB AT 206 : BOOL := false;
    manufacturing/syrup/arrivalValveSyrup1/cmdOfValve/faults1/openedSensorFB AT 207 : BOOL := false;
    manufacturing/syrup/arrivalValveSyrup1/cmdOfValve/faults1/acknowledgePB AT 12 : BOOL := false;
    manufacturing/syrup/arrivalValveSyrup1/cmdOfValve/faults1/generalFault AT 216 : BOOL := false;
    manufacturing/syrup/arrivalValveSyrup1/cmdOfValve/faults1/closedSensorFault AT 280 : BOOL := false;
    manufacturing/syrup/arrivalValveSyrup1/cmdOfValve/faults1/openedSensorFault AT 281 : BOOL := false;
    manufacturing/syrup/arrivalValveSyrup1/cmdOfValve/faults1/discordanceFault AT 282 : BOOL := false;
    manufacturing/syrup/arrivalValveSyrup1/cmdOfValve/faults1/presetMvt AT 677 : TIME := T#0h0m4s0ms;
    manufacturing/syrup/arrivalValveSyrup1/cmdOfValve/faults1/presetDiscordance AT 681 : TIME := T#0h0m0s200ms;
    manufacturing/syrup/arrivalValveSyrup1/valve/voltage380 AT 272 : BOOL := true;
    manufacturing/syrup/arrivalValveSyrup1/valve/cmdSupply AT 271 : BOOL := true;
    manufacturing/syrup/arrivalValveSyrup1/valve/sensorSupply AT 270 : BOOL := true;
    manufacturing/syrup/arrivalValveSyrup1/valve/openCmd AT 275 : BOOL := false;
    manufacturing/syrup/arrivalValveSyrup1/valve/closeCmd AT 276 : BOOL := false;
    manufacturing/syrup/arrivalValveSyrup1/valve/inputFlow AT 96 : REAL := 50.0;
    manufacturing/syrup/arrivalValveSyrup1/valve/openedSensor AT 207 : BOOL := false;
    manufacturing/syrup/arrivalValveSyrup1/valve/closedSensor AT 206 : BOOL := false;
    manufacturing/syrup/arrivalValveSyrup1/valve/outputFlow AT 99 : REAL := 0.0;
    manufacturing/syrup/arrivalValveSyrup1/valve/percentOpening AT 95 : REAL := 0.0;
    manufacturing/syrup/arrivalValveSyrup1/valve/increment AT 109 : REAL := 0.0;
    manufacturing/syrup/arrivalValveSyrup1/valve/memoOpen AT 292 : BOOL := false;
    manufacturing/syrup/arrivalValveSyrup1/valve/memoClose AT 293 : BOOL := false;
    manufacturing/syrup/arrivalValveSyrup1/valve/openState AT 294 : BOOL := false;
    manufacturing/syrup/arrivalValveSyrup1/valve/closeState AT 295 : BOOL := false;
    manufacturing/syrup/arrivalValveSyrup1/valve/openingVal AT 110 : REAL := 0.0;
    manufacturing/syrup/arrivalValveSyrup1/valve/unit AT 111 : REAL := 0.0;
    manufacturing/syrup/arrivalValveSyrup1/valve/openingTime AT 112 : REAL := 0.5;
    manufacturing/syrup/arrivalValveSyrup1/valve/openedSensorLogic AT 296 : BOOL := true;
    manufacturing/syrup/arrivalValveSyrup1/valve/closedSensorLogic AT 297 : BOOL := true;
    manufacturing/syrup/arrivalValveSyrup1/valve/flowMax AT 113 : REAL := 10000.0;
    manufacturing/syrup/arrivalValveSyrup1/valve/flowPerHour AT 298 : BOOL := true;
    manufacturing/syrup/arrivalValveSyrup1/valve/flowPerMinute AT 299 : BOOL := false;
    manufacturing/syrup/arrivalValveSyrup1/valve/d_locking AT 300 : BOOL := false;
    manufacturing/syrup/arrivalValveSyrup1/valve/v_d_locking AT 114 : REAL := 2.0;
    manufacturing/syrup/arrivalValveSyrup1/valve/d_flow AT 301 : BOOL := false;
    manufacturing/syrup/arrivalValveSyrup1/valve/v_d_flow AT 115 : REAL := 2.0;
    manufacturing/syrup/arrivalValveSyrup1/valve/d_electrical AT 302 : BOOL := false;
    manufacturing/syrup/arrivalValveSyrup1/valve/v_d_electrical AT 303 : BOOL := false;
    manufacturing/syrup/arrivalValveSyrup1/valve/d_closedSensor AT 304 : BOOL := false;
    manufacturing/syrup/arrivalValveSyrup1/valve/v_d_closedSensor AT 305 : BOOL := false;
    manufacturing/syrup/arrivalValveSyrup1/valve/d_openedSensor AT 306 : BOOL := false;
    manufacturing/syrup/arrivalValveSyrup1/valve/v_d_openedSensor AT 307 : BOOL := false;
    manufacturing/syrup/arrivalValveSyrup2/acknowledgePB AT 12 : BOOL := false;
    manufacturing/syrup/arrivalValveSyrup2/autoMode AT 23 : BOOL := false;
    manufacturing/syrup/arrivalValveSyrup2/manualMode AT 24 : BOOL := false;
    manufacturing/syrup/arrivalValveSyrup2/autoCloseCmd AT 210 : BOOL := false;
    manufacturing/syrup/arrivalValveSyrup2/autoOpenCmd AT 211 : BOOL := false;
    manufacturing/syrup/arrivalValveSyrup2/inputFlow AT 94 : REAL := 50.0;
    manufacturing/syrup/arrivalValveSyrup2/openedSensor AT 205 : BOOL := false;
    manufacturing/syrup/arrivalValveSyrup2/closedSensor AT 204 : BOOL := false;
    manufacturing/syrup/arrivalValveSyrup2/generalFault AT 217 : BOOL := false;
    manufacturing/syrup/arrivalValveSyrup2/outputFlow AT 100 : REAL := 0.0;
    manufacturing/syrup/arrivalValveSyrup2/percentOpening AT 93 : REAL := 0.0;
    manufacturing/syrup/arrivalValveSyrup2/panel1/closeValvePB AT 311 : BOOL := false;
    manufacturing/syrup/arrivalValveSyrup2/panel1/openValvePB AT 312 : BOOL := false;
    manufacturing/syrup/arrivalValveSyrup2/panel1/switch/leftVariable AT 311 : BOOL := false;
    manufacturing/syrup/arrivalValveSyrup2/panel1/switch/rightVariable AT 312 : BOOL := false;
    manufacturing/syrup/arrivalValveSyrup2/panel1/switch/leftPosition AT 315 : BOOL := false;
    manufacturing/syrup/arrivalValveSyrup2/panel1/switch/middlePosition AT 316 : BOOL := false;
    manufacturing/syrup/arrivalValveSyrup2/panel1/switch/rightPosition AT 317 : BOOL := false;
    manufacturing/syrup/arrivalValveSyrup2/cmdOfValve/autoMode AT 23 : BOOL := false;
    manufacturing/syrup/arrivalValveSyrup2/cmdOfValve/manualMode AT 24 : BOOL := false;
    manufacturing/syrup/arrivalValveSyrup2/cmdOfValve/closedSensorFB AT 204 : BOOL := false;
    manufacturing/syrup/arrivalValveSyrup2/cmdOfValve/openedSensorFB AT 205 : BOOL := false;
    manufacturing/syrup/arrivalValveSyrup2/cmdOfValve/autoCloseCmd AT 210 : BOOL := false;
    manufacturing/syrup/arrivalValveSyrup2/cmdOfValve/autoOpenCmd AT 211 : BOOL := false;
    manufacturing/syrup/arrivalValveSyrup2/cmdOfValve/closeValvePB AT 311 : BOOL := false;
    manufacturing/syrup/arrivalValveSyrup2/cmdOfValve/openValvePB AT 312 : BOOL := false;
    manufacturing/syrup/arrivalValveSyrup2/cmdOfValve/acknowledgePB AT 12 : BOOL := false;
    manufacturing/syrup/arrivalValveSyrup2/cmdOfValve/closeCmd AT 314 : BOOL := false;
    manufacturing/syrup/arrivalValveSyrup2/cmdOfValve/openCmd AT 313 : BOOL := false;
    manufacturing/syrup/arrivalValveSyrup2/cmdOfValve/generalFault AT 217 : BOOL := false;
    manufacturing/syrup/arrivalValveSyrup2/cmdOfValve/actions/autoMode AT 23 : BOOL := false;
    manufacturing/syrup/arrivalValveSyrup2/cmdOfValve/actions/manualMode AT 24 : BOOL := false;
    manufacturing/syrup/arrivalValveSyrup2/cmdOfValve/actions/autoCloseCmd AT 210 : BOOL := false;
    manufacturing/syrup/arrivalValveSyrup2/cmdOfValve/actions/autoOpenCmd AT 211 : BOOL := false;
    manufacturing/syrup/arrivalValveSyrup2/cmdOfValve/actions/closedSensorFB AT 204 : BOOL := false;
    manufacturing/syrup/arrivalValveSyrup2/cmdOfValve/actions/openedSensorFB AT 205 : BOOL := false;
    manufacturing/syrup/arrivalValveSyrup2/cmdOfValve/actions/closeValvePB AT 311 : BOOL := false;
    manufacturing/syrup/arrivalValveSyrup2/cmdOfValve/actions/openValvePB AT 312 : BOOL := false;
    manufacturing/syrup/arrivalValveSyrup2/cmdOfValve/actions/generalFault AT 217 : BOOL := false;
    manufacturing/syrup/arrivalValveSyrup2/cmdOfValve/actions/closeCmd AT 314 : BOOL := false;
    manufacturing/syrup/arrivalValveSyrup2/cmdOfValve/actions/openCmd AT 313 : BOOL := false;
    manufacturing/syrup/arrivalValveSyrup2/cmdOfValve/faults1/closeCmd AT 314 : BOOL := false;
    manufacturing/syrup/arrivalValveSyrup2/cmdOfValve/faults1/openCmd AT 313 : BOOL := false;
    manufacturing/syrup/arrivalValveSyrup2/cmdOfValve/faults1/closedSensorFB AT 204 : BOOL := false;
    manufacturing/syrup/arrivalValveSyrup2/cmdOfValve/faults1/openedSensorFB AT 205 : BOOL := false;
    manufacturing/syrup/arrivalValveSyrup2/cmdOfValve/faults1/acknowledgePB AT 12 : BOOL := false;
    manufacturing/syrup/arrivalValveSyrup2/cmdOfValve/faults1/generalFault AT 217 : BOOL := false;
    manufacturing/syrup/arrivalValveSyrup2/cmdOfValve/faults1/closedSensorFault AT 318 : BOOL := false;
    manufacturing/syrup/arrivalValveSyrup2/cmdOfValve/faults1/openedSensorFault AT 319 : BOOL := false;
    manufacturing/syrup/arrivalValveSyrup2/cmdOfValve/faults1/discordanceFault AT 320 : BOOL := false;
    manufacturing/syrup/arrivalValveSyrup2/cmdOfValve/faults1/presetMvt AT 718 : TIME := T#0h0m4s0ms;
    manufacturing/syrup/arrivalValveSyrup2/cmdOfValve/faults1/presetDiscordance AT 722 : TIME := T#0h0m0s200ms;
    manufacturing/syrup/arrivalValveSyrup2/valve/voltage380 AT 310 : BOOL := true;
    manufacturing/syrup/arrivalValveSyrup2/valve/cmdSupply AT 309 : BOOL := true;
    manufacturing/syrup/arrivalValveSyrup2/valve/sensorSupply AT 308 : BOOL := true;
    manufacturing/syrup/arrivalValveSyrup2/valve/openCmd AT 313 : BOOL := false;
    manufacturing/syrup/arrivalValveSyrup2/valve/closeCmd AT 314 : BOOL := false;
    manufacturing/syrup/arrivalValveSyrup2/valve/inputFlow AT 94 : REAL := 50.0;
    manufacturing/syrup/arrivalValveSyrup2/valve/openedSensor AT 205 : BOOL := false;
    manufacturing/syrup/arrivalValveSyrup2/valve/closedSensor AT 204 : BOOL := false;
    manufacturing/syrup/arrivalValveSyrup2/valve/outputFlow AT 100 : REAL := 0.0;
    manufacturing/syrup/arrivalValveSyrup2/valve/percentOpening AT 93 : REAL := 0.0;
    manufacturing/syrup/arrivalValveSyrup2/valve/increment AT 119 : REAL := 0.0;
    manufacturing/syrup/arrivalValveSyrup2/valve/memoOpen AT 330 : BOOL := false;
    manufacturing/syrup/arrivalValveSyrup2/valve/memoClose AT 331 : BOOL := false;
    manufacturing/syrup/arrivalValveSyrup2/valve/openState AT 332 : BOOL := false;
    manufacturing/syrup/arrivalValveSyrup2/valve/closeState AT 333 : BOOL := false;
    manufacturing/syrup/arrivalValveSyrup2/valve/openingVal AT 120 : REAL := 0.0;
    manufacturing/syrup/arrivalValveSyrup2/valve/unit AT 121 : REAL := 0.0;
    manufacturing/syrup/arrivalValveSyrup2/valve/openingTime AT 122 : REAL := 0.5;
    manufacturing/syrup/arrivalValveSyrup2/valve/openedSensorLogic AT 334 : BOOL := true;
    manufacturing/syrup/arrivalValveSyrup2/valve/closedSensorLogic AT 335 : BOOL := true;
    manufacturing/syrup/arrivalValveSyrup2/valve/flowMax AT 123 : REAL := 10000.0;
    manufacturing/syrup/arrivalValveSyrup2/valve/flowPerHour AT 336 : BOOL := true;
    manufacturing/syrup/arrivalValveSyrup2/valve/flowPerMinute AT 337 : BOOL := false;
    manufacturing/syrup/arrivalValveSyrup2/valve/d_locking AT 338 : BOOL := false;
    manufacturing/syrup/arrivalValveSyrup2/valve/v_d_locking AT 124 : REAL := 2.0;
    manufacturing/syrup/arrivalValveSyrup2/valve/d_flow AT 339 : BOOL := false;
    manufacturing/syrup/arrivalValveSyrup2/valve/v_d_flow AT 125 : REAL := 2.0;
    manufacturing/syrup/arrivalValveSyrup2/valve/d_electrical AT 340 : BOOL := false;
    manufacturing/syrup/arrivalValveSyrup2/valve/v_d_electrical AT 341 : BOOL := false;
    manufacturing/syrup/arrivalValveSyrup2/valve/d_closedSensor AT 342 : BOOL := false;
    manufacturing/syrup/arrivalValveSyrup2/valve/v_d_closedSensor AT 343 : BOOL := false;
    manufacturing/syrup/arrivalValveSyrup2/valve/d_openedSensor AT 344 : BOOL := false;
    manufacturing/syrup/arrivalValveSyrup2/valve/v_d_openedSensor AT 345 : BOOL := false;
    manufacturing/syrup/arrivalValveSyrup3/acknowledgePB AT 12 : BOOL := false;
    manufacturing/syrup/arrivalValveSyrup3/autoMode AT 23 : BOOL := false;
    manufacturing/syrup/arrivalValveSyrup3/manualMode AT 24 : BOOL := false;
    manufacturing/syrup/arrivalValveSyrup3/autoCloseCmd AT 212 : BOOL := false;
    manufacturing/syrup/arrivalValveSyrup3/autoOpenCmd AT 213 : BOOL := false;
    manufacturing/syrup/arrivalValveSyrup3/inputFlow AT 92 : REAL := 50.0;
    manufacturing/syrup/arrivalValveSyrup3/openedSensor AT 203 : BOOL := false;
    manufacturing/syrup/arrivalValveSyrup3/closedSensor AT 202 : BOOL := false;
    manufacturing/syrup/arrivalValveSyrup3/generalFault AT 218 : BOOL := false;
    manufacturing/syrup/arrivalValveSyrup3/outputFlow AT 101 : REAL := 0.0;
    manufacturing/syrup/arrivalValveSyrup3/percentOpening AT 91 : REAL := 0.0;
    manufacturing/syrup/arrivalValveSyrup3/panel1/closeValvePB AT 349 : BOOL := false;
    manufacturing/syrup/arrivalValveSyrup3/panel1/openValvePB AT 350 : BOOL := false;
    manufacturing/syrup/arrivalValveSyrup3/panel1/switch/leftVariable AT 349 : BOOL := false;
    manufacturing/syrup/arrivalValveSyrup3/panel1/switch/rightVariable AT 350 : BOOL := false;
    manufacturing/syrup/arrivalValveSyrup3/panel1/switch/leftPosition AT 353 : BOOL := false;
    manufacturing/syrup/arrivalValveSyrup3/panel1/switch/middlePosition AT 354 : BOOL := false;
    manufacturing/syrup/arrivalValveSyrup3/panel1/switch/rightPosition AT 355 : BOOL := false;
    manufacturing/syrup/arrivalValveSyrup3/cmdOfValve/autoMode AT 23 : BOOL := false;
    manufacturing/syrup/arrivalValveSyrup3/cmdOfValve/manualMode AT 24 : BOOL := false;
    manufacturing/syrup/arrivalValveSyrup3/cmdOfValve/closedSensorFB AT 202 : BOOL := false;
    manufacturing/syrup/arrivalValveSyrup3/cmdOfValve/openedSensorFB AT 203 : BOOL := false;
    manufacturing/syrup/arrivalValveSyrup3/cmdOfValve/autoCloseCmd AT 212 : BOOL := false;
    manufacturing/syrup/arrivalValveSyrup3/cmdOfValve/autoOpenCmd AT 213 : BOOL := false;
    manufacturing/syrup/arrivalValveSyrup3/cmdOfValve/closeValvePB AT 349 : BOOL := false;
    manufacturing/syrup/arrivalValveSyrup3/cmdOfValve/openValvePB AT 350 : BOOL := false;
    manufacturing/syrup/arrivalValveSyrup3/cmdOfValve/acknowledgePB AT 12 : BOOL := false;
    manufacturing/syrup/arrivalValveSyrup3/cmdOfValve/closeCmd AT 352 : BOOL := false;
    manufacturing/syrup/arrivalValveSyrup3/cmdOfValve/openCmd AT 351 : BOOL := false;
    manufacturing/syrup/arrivalValveSyrup3/cmdOfValve/generalFault AT 218 : BOOL := false;
    manufacturing/syrup/arrivalValveSyrup3/cmdOfValve/actions/autoMode AT 23 : BOOL := false;
    manufacturing/syrup/arrivalValveSyrup3/cmdOfValve/actions/manualMode AT 24 : BOOL := false;
    manufacturing/syrup/arrivalValveSyrup3/cmdOfValve/actions/autoCloseCmd AT 212 : BOOL := false;
    manufacturing/syrup/arrivalValveSyrup3/cmdOfValve/actions/autoOpenCmd AT 213 : BOOL := false;
    manufacturing/syrup/arrivalValveSyrup3/cmdOfValve/actions/closedSensorFB AT 202 : BOOL := false;
    manufacturing/syrup/arrivalValveSyrup3/cmdOfValve/actions/openedSensorFB AT 203 : BOOL := false;
    manufacturing/syrup/arrivalValveSyrup3/cmdOfValve/actions/closeValvePB AT 349 : BOOL := false;
    manufacturing/syrup/arrivalValveSyrup3/cmdOfValve/actions/openValvePB AT 350 : BOOL := false;
    manufacturing/syrup/arrivalValveSyrup3/cmdOfValve/actions/generalFault AT 218 : BOOL := false;
    manufacturing/syrup/arrivalValveSyrup3/cmdOfValve/actions/closeCmd AT 352 : BOOL := false;
    manufacturing/syrup/arrivalValveSyrup3/cmdOfValve/actions/openCmd AT 351 : BOOL := false;
    manufacturing/syrup/arrivalValveSyrup3/cmdOfValve/faults1/closeCmd AT 352 : BOOL := false;
    manufacturing/syrup/arrivalValveSyrup3/cmdOfValve/faults1/openCmd AT 351 : BOOL := false;
    manufacturing/syrup/arrivalValveSyrup3/cmdOfValve/faults1/closedSensorFB AT 202 : BOOL := false;
    manufacturing/syrup/arrivalValveSyrup3/cmdOfValve/faults1/openedSensorFB AT 203 : BOOL := false;
    manufacturing/syrup/arrivalValveSyrup3/cmdOfValve/faults1/acknowledgePB AT 12 : BOOL := false;
    manufacturing/syrup/arrivalValveSyrup3/cmdOfValve/faults1/generalFault AT 218 : BOOL := false;
    manufacturing/syrup/arrivalValveSyrup3/cmdOfValve/faults1/closedSensorFault AT 356 : BOOL := false;
    manufacturing/syrup/arrivalValveSyrup3/cmdOfValve/faults1/openedSensorFault AT 357 : BOOL := false;
    manufacturing/syrup/arrivalValveSyrup3/cmdOfValve/faults1/discordanceFault AT 358 : BOOL := false;
    manufacturing/syrup/arrivalValveSyrup3/cmdOfValve/faults1/presetMvt AT 759 : TIME := T#0h0m4s0ms;
    manufacturing/syrup/arrivalValveSyrup3/cmdOfValve/faults1/presetDiscordance AT 763 : TIME := T#0h0m0s200ms;
    manufacturing/syrup/arrivalValveSyrup3/valve/voltage380 AT 348 : BOOL := true;
    manufacturing/syrup/arrivalValveSyrup3/valve/cmdSupply AT 347 : BOOL := true;
    manufacturing/syrup/arrivalValveSyrup3/valve/sensorSupply AT 346 : BOOL := true;
    manufacturing/syrup/arrivalValveSyrup3/valve/openCmd AT 351 : BOOL := false;
    manufacturing/syrup/arrivalValveSyrup3/valve/closeCmd AT 352 : BOOL := false;
    manufacturing/syrup/arrivalValveSyrup3/valve/inputFlow AT 92 : REAL := 50.0;
    manufacturing/syrup/arrivalValveSyrup3/valve/openedSensor AT 203 : BOOL := false;
    manufacturing/syrup/arrivalValveSyrup3/valve/closedSensor AT 202 : BOOL := false;
    manufacturing/syrup/arrivalValveSyrup3/valve/outputFlow AT 101 : REAL := 0.0;
    manufacturing/syrup/arrivalValveSyrup3/valve/percentOpening AT 91 : REAL := 0.0;
    manufacturing/syrup/arrivalValveSyrup3/valve/increment AT 129 : REAL := 0.0;
    manufacturing/syrup/arrivalValveSyrup3/valve/memoOpen AT 368 : BOOL := false;
    manufacturing/syrup/arrivalValveSyrup3/valve/memoClose AT 369 : BOOL := false;
    manufacturing/syrup/arrivalValveSyrup3/valve/openState AT 370 : BOOL := false;
    manufacturing/syrup/arrivalValveSyrup3/valve/closeState AT 371 : BOOL := false;
    manufacturing/syrup/arrivalValveSyrup3/valve/openingVal AT 130 : REAL := 0.0;
    manufacturing/syrup/arrivalValveSyrup3/valve/unit AT 131 : REAL := 0.0;
    manufacturing/syrup/arrivalValveSyrup3/valve/openingTime AT 132 : REAL := 0.5;
    manufacturing/syrup/arrivalValveSyrup3/valve/openedSensorLogic AT 372 : BOOL := true;
    manufacturing/syrup/arrivalValveSyrup3/valve/closedSensorLogic AT 373 : BOOL := true;
    manufacturing/syrup/arrivalValveSyrup3/valve/flowMax AT 133 : REAL := 10000.0;
    manufacturing/syrup/arrivalValveSyrup3/valve/flowPerHour AT 374 : BOOL := true;
    manufacturing/syrup/arrivalValveSyrup3/valve/flowPerMinute AT 375 : BOOL := false;
    manufacturing/syrup/arrivalValveSyrup3/valve/d_locking AT 376 : BOOL := false;
    manufacturing/syrup/arrivalValveSyrup3/valve/v_d_locking AT 134 : REAL := 2.0;
    manufacturing/syrup/arrivalValveSyrup3/valve/d_flow AT 377 : BOOL := false;
    manufacturing/syrup/arrivalValveSyrup3/valve/v_d_flow AT 135 : REAL := 2.0;
    manufacturing/syrup/arrivalValveSyrup3/valve/d_electrical AT 378 : BOOL := false;
    manufacturing/syrup/arrivalValveSyrup3/valve/v_d_electrical AT 379 : BOOL := false;
    manufacturing/syrup/arrivalValveSyrup3/valve/d_closedSensor AT 380 : BOOL := false;
    manufacturing/syrup/arrivalValveSyrup3/valve/v_d_closedSensor AT 381 : BOOL := false;
    manufacturing/syrup/arrivalValveSyrup3/valve/d_openedSensor AT 382 : BOOL := false;
    manufacturing/syrup/arrivalValveSyrup3/valve/v_d_openedSensor AT 383 : BOOL := false;
    manufacturing/syrup/syrupExtractionValve/acknowledgePB AT 12 : BOOL := false;
    manufacturing/syrup/syrupExtractionValve/autoMode AT 23 : BOOL := false;
    manufacturing/syrup/syrupExtractionValve/manualMode AT 24 : BOOL := false;
    manufacturing/syrup/syrupExtractionValve/autoCloseCmd AT 214 : BOOL := false;
    manufacturing/syrup/syrupExtractionValve/autoOpenCmd AT 215 : BOOL := false;
    manufacturing/syrup/syrupExtractionValve/inputFlow AT 98 : REAL := 0.0;
    manufacturing/syrup/syrupExtractionValve/openedSensor AT 201 : BOOL := false;
    manufacturing/syrup/syrupExtractionValve/closedSensor AT 200 : BOOL := false;
    manufacturing/syrup/syrupExtractionValve/generalFault AT 219 : BOOL := false;
    manufacturing/syrup/syrupExtractionValve/outputFlow AT 27 : REAL := 0.0;
    manufacturing/syrup/syrupExtractionValve/percentOpening AT 90 : REAL := 0.0;
    manufacturing/syrup/syrupExtractionValve/panel1/closeValvePB AT 387 : BOOL := false;
    manufacturing/syrup/syrupExtractionValve/panel1/openValvePB AT 388 : BOOL := false;
    manufacturing/syrup/syrupExtractionValve/panel1/switch/leftVariable AT 387 : BOOL := false;
    manufacturing/syrup/syrupExtractionValve/panel1/switch/rightVariable AT 388 : BOOL := false;
    manufacturing/syrup/syrupExtractionValve/panel1/switch/leftPosition AT 391 : BOOL := false;
    manufacturing/syrup/syrupExtractionValve/panel1/switch/middlePosition AT 392 : BOOL := false;
    manufacturing/syrup/syrupExtractionValve/panel1/switch/rightPosition AT 393 : BOOL := false;
    manufacturing/syrup/syrupExtractionValve/cmdOfValve/autoMode AT 23 : BOOL := false;
    manufacturing/syrup/syrupExtractionValve/cmdOfValve/manualMode AT 24 : BOOL := false;
    manufacturing/syrup/syrupExtractionValve/cmdOfValve/closedSensorFB AT 200 : BOOL := false;
    manufacturing/syrup/syrupExtractionValve/cmdOfValve/openedSensorFB AT 201 : BOOL := false;
    manufacturing/syrup/syrupExtractionValve/cmdOfValve/autoCloseCmd AT 214 : BOOL := false;
    manufacturing/syrup/syrupExtractionValve/cmdOfValve/autoOpenCmd AT 215 : BOOL := false;
    manufacturing/syrup/syrupExtractionValve/cmdOfValve/closeValvePB AT 387 : BOOL := false;
    manufacturing/syrup/syrupExtractionValve/cmdOfValve/openValvePB AT 388 : BOOL := false;
    manufacturing/syrup/syrupExtractionValve/cmdOfValve/acknowledgePB AT 12 : BOOL := false;
    manufacturing/syrup/syrupExtractionValve/cmdOfValve/closeCmd AT 390 : BOOL := false;
    manufacturing/syrup/syrupExtractionValve/cmdOfValve/openCmd AT 389 : BOOL := false;
    manufacturing/syrup/syrupExtractionValve/cmdOfValve/generalFault AT 219 : BOOL := false;
    manufacturing/syrup/syrupExtractionValve/cmdOfValve/actions/autoMode AT 23 : BOOL := false;
    manufacturing/syrup/syrupExtractionValve/cmdOfValve/actions/manualMode AT 24 : BOOL := false;
    manufacturing/syrup/syrupExtractionValve/cmdOfValve/actions/autoCloseCmd AT 214 : BOOL := false;
    manufacturing/syrup/syrupExtractionValve/cmdOfValve/actions/autoOpenCmd AT 215 : BOOL := false;
    manufacturing/syrup/syrupExtractionValve/cmdOfValve/actions/closedSensorFB AT 200 : BOOL := false;
    manufacturing/syrup/syrupExtractionValve/cmdOfValve/actions/openedSensorFB AT 201 : BOOL := false;
    manufacturing/syrup/syrupExtractionValve/cmdOfValve/actions/closeValvePB AT 387 : BOOL := false;
    manufacturing/syrup/syrupExtractionValve/cmdOfValve/actions/openValvePB AT 388 : BOOL := false;
    manufacturing/syrup/syrupExtractionValve/cmdOfValve/actions/generalFault AT 219 : BOOL := false;
    manufacturing/syrup/syrupExtractionValve/cmdOfValve/actions/closeCmd AT 390 : BOOL := false;
    manufacturing/syrup/syrupExtractionValve/cmdOfValve/actions/openCmd AT 389 : BOOL := false;
    manufacturing/syrup/syrupExtractionValve/cmdOfValve/faults1/closeCmd AT 390 : BOOL := false;
    manufacturing/syrup/syrupExtractionValve/cmdOfValve/faults1/openCmd AT 389 : BOOL := false;
    manufacturing/syrup/syrupExtractionValve/cmdOfValve/faults1/closedSensorFB AT 200 : BOOL := false;
    manufacturing/syrup/syrupExtractionValve/cmdOfValve/faults1/openedSensorFB AT 201 : BOOL := false;
    manufacturing/syrup/syrupExtractionValve/cmdOfValve/faults1/acknowledgePB AT 12 : BOOL := false;
    manufacturing/syrup/syrupExtractionValve/cmdOfValve/faults1/generalFault AT 219 : BOOL := false;
    manufacturing/syrup/syrupExtractionValve/cmdOfValve/faults1/closedSensorFault AT 394 : BOOL := false;
    manufacturing/syrup/syrupExtractionValve/cmdOfValve/faults1/openedSensorFault AT 395 : BOOL := false;
    manufacturing/syrup/syrupExtractionValve/cmdOfValve/faults1/discordanceFault AT 396 : BOOL := false;
    manufacturing/syrup/syrupExtractionValve/cmdOfValve/faults1/presetMvt AT 800 : TIME := T#0h0m4s0ms;
    manufacturing/syrup/syrupExtractionValve/cmdOfValve/faults1/presetDiscordance AT 804 : TIME := T#0h0m0s200ms;
    manufacturing/syrup/syrupExtractionValve/valve/voltage380 AT 386 : BOOL := true;
    manufacturing/syrup/syrupExtractionValve/valve/cmdSupply AT 385 : BOOL := true;
    manufacturing/syrup/syrupExtractionValve/valve/sensorSupply AT 384 : BOOL := true;
    manufacturing/syrup/syrupExtractionValve/valve/openCmd AT 389 : BOOL := false;
    manufacturing/syrup/syrupExtractionValve/valve/closeCmd AT 390 : BOOL := false;
    manufacturing/syrup/syrupExtractionValve/valve/inputFlow AT 98 : REAL := 0.0;
    manufacturing/syrup/syrupExtractionValve/valve/openedSensor AT 201 : BOOL := false;
    manufacturing/syrup/syrupExtractionValve/valve/closedSensor AT 200 : BOOL := false;
    manufacturing/syrup/syrupExtractionValve/valve/outputFlow AT 27 : REAL := 0.0;
    manufacturing/syrup/syrupExtractionValve/valve/percentOpening AT 90 : REAL := 0.0;
    manufacturing/syrup/syrupExtractionValve/valve/increment AT 139 : REAL := 0.0;
    manufacturing/syrup/syrupExtractionValve/valve/memoOpen AT 406 : BOOL := false;
    manufacturing/syrup/syrupExtractionValve/valve/memoClose AT 407 : BOOL := false;
    manufacturing/syrup/syrupExtractionValve/valve/openState AT 408 : BOOL := false;
    manufacturing/syrup/syrupExtractionValve/valve/closeState AT 409 : BOOL := false;
    manufacturing/syrup/syrupExtractionValve/valve/openingVal AT 140 : REAL := 0.0;
    manufacturing/syrup/syrupExtractionValve/valve/unit AT 141 : REAL := 0.0;
    manufacturing/syrup/syrupExtractionValve/valve/openingTime AT 142 : REAL := 0.5;
    manufacturing/syrup/syrupExtractionValve/valve/openedSensorLogic AT 410 : BOOL := true;
    manufacturing/syrup/syrupExtractionValve/valve/closedSensorLogic AT 411 : BOOL := true;
    manufacturing/syrup/syrupExtractionValve/valve/flowMax AT 143 : REAL := 10000.0;
    manufacturing/syrup/syrupExtractionValve/valve/flowPerHour AT 412 : BOOL := true;
    manufacturing/syrup/syrupExtractionValve/valve/flowPerMinute AT 413 : BOOL := false;
    manufacturing/syrup/syrupExtractionValve/valve/d_locking AT 414 : BOOL := false;
    manufacturing/syrup/syrupExtractionValve/valve/v_d_locking AT 144 : REAL := 2.0;
    manufacturing/syrup/syrupExtractionValve/valve/d_flow AT 415 : BOOL := false;
    manufacturing/syrup/syrupExtractionValve/valve/v_d_flow AT 145 : REAL := 2.0;
    manufacturing/syrup/syrupExtractionValve/valve/d_electrical AT 416 : BOOL := false;
    manufacturing/syrup/syrupExtractionValve/valve/v_d_electrical AT 417 : BOOL := false;
    manufacturing/syrup/syrupExtractionValve/valve/d_closedSensor AT 418 : BOOL := false;
    manufacturing/syrup/syrupExtractionValve/valve/v_d_closedSensor AT 419 : BOOL := false;
    manufacturing/syrup/syrupExtractionValve/valve/d_openedSensor AT 420 : BOOL := false;
    manufacturing/syrup/syrupExtractionValve/valve/v_d_openedSensor AT 421 : BOOL := false;
    manufacturing/syrup/faults1/generalFault1 AT 216 : BOOL := false;
    manufacturing/syrup/faults1/generalFault2 AT 217 : BOOL := false;
    manufacturing/syrup/faults1/generalFault3 AT 218 : BOOL := false;
    manufacturing/syrup/faults1/generalFault4 AT 219 : BOOL := false;
    manufacturing/syrup/faults1/fault AT 54 : BOOL := false;
    manufacturing/syrup/syrupQuantity/flowSyrup1 AT 99 : REAL := 0.0;
    manufacturing/syrup/syrupQuantity/flowSyrup2 AT 100 : REAL := 0.0;
    manufacturing/syrup/syrupQuantity/flowSyrup3 AT 101 : REAL := 0.0;
    manufacturing/syrup/syrupQuantity/flow AT 102 : REAL := 0.0;
    manufacturing/syrup/syrupsTank/inletFlow AT 102 : REAL := 0.0;
    manufacturing/syrup/syrupsTank/outletFlow AT 27 : REAL := 0.0;
    manufacturing/syrup/syrupsTank/tankLevel AT 97 : REAL := 0.0;
    manufacturing/syrup/syrupsTank/percent AT 146 : REAL := 0.0;
    manufacturing/syrup/syrupsTank/capacity AT 147 : REAL := 300.0;
    manufacturing/syrup/syrupsTank/d_level AT 422 : BOOL := false;
    manufacturing/syrup/syrupsTank/v_d_level AT 148 : REAL := 0.0;
    manufacturing/syrup/level/measure AT 97 : REAL := 0.0;
    manufacturing/syrup/level/sensorSupply AT 199 : BOOL := true;
    manufacturing/syrup/level/realValue AT 103 : REAL := 0.0;
    manufacturing/syrup/level/intValue AT 89 : REAL := 0.0;
    manufacturing/syrup/level/dintValue AT 88 : REAL := 0.0;
    manufacturing/syrup/level/tmp AT 832 : DINT := 0;
    manufacturing/syrup/level/localValue AT 149 : REAL := 0.0;
    manufacturing/syrup/level/nbDigit AT 833 : SINT := 2;
    manufacturing/syrup/level/d_value AT 423 : BOOL := false;
    manufacturing/syrup/level/v_d_value AT 150 : REAL := 0.0;
    manufacturing/syrup/scale/inputValue AT 103 : REAL := 0.0;
    manufacturing/syrup/scale/realValue AT 87 : REAL := 0.0;
    manufacturing/syrup/scale/dintValue AT 662 : DINT := 0;
    manufacturing/syrup/scale/intValue AT 661 : INT := 0;
    manufacturing/syrup/scale/a AT 151 : REAL := 0.0;
    manufacturing/syrup/scale/b AT 152 : REAL := 0.0;
    manufacturing/syrup/scale/k AT 153 : REAL := 0.0;
    manufacturing/syrup/scale/minInput AT 154 : REAL := 0.0;
    manufacturing/syrup/scale/maxInput AT 155 : REAL := 300.0;
    manufacturing/syrup/scale/minOutput AT 156 : REAL := 0.0;
    manufacturing/syrup/scale/maxOutput AT 157 : REAL := 300.0;
    manufacturing/syrup/scale/d_scale AT 424 : BOOL := false;
    manufacturing/syrup/scale/v_d_scale AT 158 : REAL := 0.0;
    manufacturing/mixture/cycleInProgress AT 15 : BOOL := false;
    manufacturing/mixture/kneadingRequest AT 22 : BOOL := false;
    manufacturing/mixture/acknowledgePB AT 12 : BOOL := false;
    manufacturing/mixture/autoMode AT 23 : BOOL := false;
    manufacturing/mixture/manualMode AT 24 : BOOL := false;
    manufacturing/mixture/syrupExtraction AT 27 : REAL := 0.0;
    manufacturing/mixture/flourExtraction AT 28 : REAL := 0.0;
    manufacturing/mixture/kneadingOK AT 17 : BOOL := false;
    manufacturing/mixture/fault AT 52 : BOOL := false;
    manufacturing/mixture/collectedMixture/flowSyrup1 AT 27 : REAL := 0.0;
    manufacturing/mixture/collectedMixture/flowSyrup2 AT 28 : REAL := 0.0;
    manufacturing/mixture/collectedMixture/flowSyrup3 AT 168 : REAL := 0.0;
    manufacturing/mixture/collectedMixture/flow AT 171 : REAL := 0.0;
    manufacturing/mixture/flow/inputFlow AT 169 : REAL := 0.0;
    manufacturing/mixture/flow/outputFlow AT 170 : REAL := 0.0;
    manufacturing/mixture/flow/unit AT 174 : REAL := 0.0;
    manufacturing/mixture/flow/flowMax AT 175 : REAL := 40000.0;
    manufacturing/mixture/flow/flowPerHour AT 438 : BOOL := true;
    manufacturing/mixture/flow/flowPerMinute AT 439 : BOOL := false;
    manufacturing/mixture/kneading/kneadingRequest AT 22 : BOOL := false;
    manufacturing/mixture/kneading/cycleInProgress AT 15 : BOOL := false;
    manufacturing/mixture/kneading/mixtureLevel AT 835 : DINT := 0;
    manufacturing/mixture/kneading/kneadingOK AT 17 : BOOL := false;
    manufacturing/mixture/kneading/knead AT 430 : BOOL := false;
    manufacturing/mixture/kneading/clean AT 432 : BOOL := false;
    manufacturing/mixture/kneading/cleaningEnd AT 431 : BOOL := false;
    manufacturing/mixture/kneading/evacuateMixture AT 434 : BOOL := false;
    manufacturing/mixture/kneading/evacMixtureEnd AT 433 : BOOL := false;
    manufacturing/mixture/kneading/nbCycles AT 836 : DINT := 0;
    manufacturing/mixture/kneading/_X_10 AT 440 : BOOL := true;
    manufacturing/mixture/kneading/_X_11 AT 441 : BOOL := false;
    manufacturing/mixture/kneading/_X_12 AT 442 : BOOL := false;
    manufacturing/mixture/kneading/_X_13 AT 443 : BOOL := false;
    manufacturing/mixture/kneading/_X_14 AT 444 : BOOL := false;
    manufacturing/mixture/kneading/_X_15 AT 445 : BOOL := false;
    manufacturing/mixture/kneading/_X_16 AT 447 : BOOL := false;
    manufacturing/mixture/kneading/_X_17 AT 446 : BOOL := false;
    manufacturing/mixture/kneading/kneadingDuration AT 837 : DINT := 20;
    manufacturing/mixture/kneading/nbOfCleanCycles AT 838 : DINT := 10;
    manufacturing/mixture/kneading/cleaningDuration AT 839 : DINT := 30;
    manufacturing/mixture/motorOfAgitator/acknowledgePB AT 12 : BOOL := false;
    manufacturing/mixture/motorOfAgitator/autoMode AT 23 : BOOL := false;
    manufacturing/mixture/motorOfAgitator/manualMode AT 24 : BOOL := false;
    manufacturing/mixture/motorOfAgitator/autoCmd AT 430 : BOOL := false;
    manufacturing/mixture/motorOfAgitator/generalFault AT 435 : BOOL := false;
    manufacturing/mixture/motorOfAgitator/speedVal AT 167 : REAL := 0.0;
    manufacturing/mixture/motorOfAgitator/speedPercent AT 166 : REAL := 0.0;
    manufacturing/mixture/motorOfAgitator/panel1/forwardPB AT 460 : BOOL := false;
    manufacturing/mixture/motorOfAgitator/panel1/stopPB AT 461 : BOOL := false;
    manufacturing/mixture/motorOfAgitator/panel1/forwardPB/PB AT 460 : BOOL := false;
    manufacturing/mixture/motorOfAgitator/panel1/forwardPB/action AT 462 : BOOL := false;
    manufacturing/mixture/motorOfAgitator/panel1/forwardPB/timeCounter AT 176 : REAL := 0.0;
    manufacturing/mixture/motorOfAgitator/panel1/forwardPB/pulseDuration AT 177 : REAL := 5.0;
    manufacturing/mixture/motorOfAgitator/panel1/forwardPB/PBLogic AT 463 : BOOL := true;
    manufacturing/mixture/motorOfAgitator/panel1/stopPB/PB AT 461 : BOOL := false;
    manufacturing/mixture/motorOfAgitator/panel1/stopPB/action AT 464 : BOOL := false;
    manufacturing/mixture/motorOfAgitator/panel1/stopPB/timeCounter AT 178 : REAL := 0.0;
    manufacturing/mixture/motorOfAgitator/panel1/stopPB/pulseDuration AT 179 : REAL := 5.0;
    manufacturing/mixture/motorOfAgitator/panel1/stopPB/PBLogic AT 465 : BOOL := true;
    manufacturing/mixture/motorOfAgitator/agitator/voltage380 AT 456 : BOOL := true;
    manufacturing/mixture/motorOfAgitator/agitator/cmdSupply AT 455 : BOOL := true;
    manufacturing/mixture/motorOfAgitator/agitator/sensorSupply AT 454 : BOOL := true;
    manufacturing/mixture/motorOfAgitator/agitator/cmd AT 457 : BOOL := false;
    manufacturing/mixture/motorOfAgitator/agitator/cmdFB AT 459 : BOOL := false;
    manufacturing/mixture/motorOfAgitator/agitator/thermal AT 458 : BOOL := false;
    manufacturing/mixture/motorOfAgitator/agitator/speedVal AT 167 : REAL := 0.0;
    manufacturing/mixture/motorOfAgitator/agitator/speedPercent AT 166 : REAL := 0.0;
    manufacturing/mixture/motorOfAgitator/agitator/increment AT 180 : REAL := 0.0;
    manufacturing/mixture/motorOfAgitator/agitator/memo AT 466 : BOOL := false;
    manufacturing/mixture/motorOfAgitator/agitator/state AT 467 : BOOL := false;
    manufacturing/mixture/motorOfAgitator/agitator/speedSetpoint AT 181 : REAL := 0.0;
    manufacturing/mixture/motorOfAgitator/agitator/cnt AT 843 : DINT := 0;
    manufacturing/mixture/motorOfAgitator/agitator/flipflop AT 468 : BOOL := false;
    manufacturing/mixture/motorOfAgitator/agitator/nominalTime AT 182 : REAL := 0.5;
    manufacturing/mixture/motorOfAgitator/agitator/thermalLogic AT 469 : BOOL := false;
    manufacturing/mixture/motorOfAgitator/agitator/cmdFbLogic AT 470 : BOOL := true;
    manufacturing/mixture/motorOfAgitator/agitator/nominalSpeed AT 183 : REAL := 5000.0;
    manufacturing/mixture/motorOfAgitator/agitator/d_locking AT 471 : BOOL := false;
    manufacturing/mixture/motorOfAgitator/agitator/v_d_locking AT 184 : REAL := 0.0;
    manufacturing/mixture/motorOfAgitator/agitator/d_electrical AT 472 : BOOL := false;
    manufacturing/mixture/motorOfAgitator/agitator/v_d_electrical AT 473 : BOOL := false;
    manufacturing/mixture/motorOfAgitator/agitator/d_cmdFB AT 474 : BOOL := false;
    manufacturing/mixture/motorOfAgitator/agitator/v_d_cmdFB AT 475 : BOOL := false;
    manufacturing/mixture/motorOfAgitator/cmdOfMotor/autoMode AT 23 : BOOL := false;
    manufacturing/mixture/motorOfAgitator/cmdOfMotor/manualMode AT 24 : BOOL := false;
    manufacturing/mixture/motorOfAgitator/cmdOfMotor/autoCmd AT 430 : BOOL := false;
    manufacturing/mixture/motorOfAgitator/cmdOfMotor/thermalFB AT 458 : BOOL := false;
    manufacturing/mixture/motorOfAgitator/cmdOfMotor/cmdFB AT 459 : BOOL := false;
    manufacturing/mixture/motorOfAgitator/cmdOfMotor/forwardPB AT 460 : BOOL := false;
    manufacturing/mixture/motorOfAgitator/cmdOfMotor/stopPB AT 461 : BOOL := false;
    manufacturing/mixture/motorOfAgitator/cmdOfMotor/acknowledgePB AT 12 : BOOL := false;
    manufacturing/mixture/motorOfAgitator/cmdOfMotor/cmd AT 457 : BOOL := false;
    manufacturing/mixture/motorOfAgitator/cmdOfMotor/generalFault AT 435 : BOOL := false;
    manufacturing/mixture/motorOfAgitator/cmdOfMotor/actions/autoMode AT 23 : BOOL := false;
    manufacturing/mixture/motorOfAgitator/cmdOfMotor/actions/manualMode AT 24 : BOOL := false;
    manufacturing/mixture/motorOfAgitator/cmdOfMotor/actions/autoCmd AT 430 : BOOL := false;
    manufacturing/mixture/motorOfAgitator/cmdOfMotor/actions/forwardPB AT 460 : BOOL := false;
    manufacturing/mixture/motorOfAgitator/cmdOfMotor/actions/stopPB AT 461 : BOOL := false;
    manufacturing/mixture/motorOfAgitator/cmdOfMotor/actions/generalFault AT 435 : BOOL := false;
    manufacturing/mixture/motorOfAgitator/cmdOfMotor/actions/cmd AT 457 : BOOL := false;
    manufacturing/mixture/motorOfAgitator/cmdOfMotor/faults1/cmd AT 457 : BOOL := false;
    manufacturing/mixture/motorOfAgitator/cmdOfMotor/faults1/thermalFB AT 458 : BOOL := false;
    manufacturing/mixture/motorOfAgitator/cmdOfMotor/faults1/cmdFB AT 459 : BOOL := false;
    manufacturing/mixture/motorOfAgitator/cmdOfMotor/faults1/acknowledgePB AT 12 : BOOL := false;
    manufacturing/mixture/motorOfAgitator/cmdOfMotor/faults1/generalFault AT 435 : BOOL := false;
    manufacturing/mixture/motorOfAgitator/cmdOfMotor/faults1/thermalFault AT 476 : BOOL := false;
    manufacturing/mixture/motorOfAgitator/cmdOfMotor/faults1/cmdFBFault AT 477 : BOOL := false;
    manufacturing/mixture/cleaningValve/acknowledgePB AT 12 : BOOL := false;
    manufacturing/mixture/cleaningValve/autoMode AT 23 : BOOL := false;
    manufacturing/mixture/cleaningValve/manualMode AT 24 : BOOL := false;
    manufacturing/mixture/cleaningValve/autoCloseCmd AT 431 : BOOL := false;
    manufacturing/mixture/cleaningValve/autoOpenCmd AT 432 : BOOL := false;
    manufacturing/mixture/cleaningValve/inputFlow AT 165 : REAL := 0.0;
    manufacturing/mixture/cleaningValve/openedSensor AT 429 : BOOL := false;
    manufacturing/mixture/cleaningValve/closedSensor AT 428 : BOOL := false;
    manufacturing/mixture/cleaningValve/generalFault AT 436 : BOOL := false;
    manufacturing/mixture/cleaningValve/outputFlow AT 164 : REAL := 0.0;
    manufacturing/mixture/cleaningValve/percentOpening AT 163 : REAL := 0.0;
    manufacturing/mixture/cleaningValve/panel1/closeValvePB AT 483 : BOOL := false;
    manufacturing/mixture/cleaningValve/panel1/openValvePB AT 484 : BOOL := false;
    manufacturing/mixture/cleaningValve/panel1/switch/leftVariable AT 483 : BOOL := false;
    manufacturing/mixture/cleaningValve/panel1/switch/rightVariable AT 484 : BOOL := false;
    manufacturing/mixture/cleaningValve/panel1/switch/leftPosition AT 487 : BOOL := false;
    manufacturing/mixture/cleaningValve/panel1/switch/middlePosition AT 488 : BOOL := false;
    manufacturing/mixture/cleaningValve/panel1/switch/rightPosition AT 489 : BOOL := false;
    manufacturing/mixture/cleaningValve/cmdOfValve/autoMode AT 23 : BOOL := false;
    manufacturing/mixture/cleaningValve/cmdOfValve/manualMode AT 24 : BOOL := false;
    manufacturing/mixture/cleaningValve/cmdOfValve/closedSensorFB AT 428 : BOOL := false;
    manufacturing/mixture/cleaningValve/cmdOfValve/openedSensorFB AT 429 : BOOL := false;
    manufacturing/mixture/cleaningValve/cmdOfValve/autoCloseCmd AT 431 : BOOL := false;
    manufacturing/mixture/cleaningValve/cmdOfValve/autoOpenCmd AT 432 : BOOL := false;
    manufacturing/mixture/cleaningValve/cmdOfValve/closeValvePB AT 483 : BOOL := false;
    manufacturing/mixture/cleaningValve/cmdOfValve/openValvePB AT 484 : BOOL := false;
    manufacturing/mixture/cleaningValve/cmdOfValve/acknowledgePB AT 12 : BOOL := false;
    manufacturing/mixture/cleaningValve/cmdOfValve/closeCmd AT 486 : BOOL := false;
    manufacturing/mixture/cleaningValve/cmdOfValve/openCmd AT 485 : BOOL := false;
    manufacturing/mixture/cleaningValve/cmdOfValve/generalFault AT 436 : BOOL := false;
    manufacturing/mixture/cleaningValve/cmdOfValve/actions/autoMode AT 23 : BOOL := false;
    manufacturing/mixture/cleaningValve/cmdOfValve/actions/manualMode AT 24 : BOOL := false;
    manufacturing/mixture/cleaningValve/cmdOfValve/actions/autoCloseCmd AT 431 : BOOL := false;
    manufacturing/mixture/cleaningValve/cmdOfValve/actions/autoOpenCmd AT 432 : BOOL := false;
    manufacturing/mixture/cleaningValve/cmdOfValve/actions/closedSensorFB AT 428 : BOOL := false;
    manufacturing/mixture/cleaningValve/cmdOfValve/actions/openedSensorFB AT 429 : BOOL := false;
    manufacturing/mixture/cleaningValve/cmdOfValve/actions/closeValvePB AT 483 : BOOL := false;
    manufacturing/mixture/cleaningValve/cmdOfValve/actions/openValvePB AT 484 : BOOL := false;
    manufacturing/mixture/cleaningValve/cmdOfValve/actions/generalFault AT 436 : BOOL := false;
    manufacturing/mixture/cleaningValve/cmdOfValve/actions/closeCmd AT 486 : BOOL := false;
    manufacturing/mixture/cleaningValve/cmdOfValve/actions/openCmd AT 485 : BOOL := false;
    manufacturing/mixture/cleaningValve/cmdOfValve/faults1/closeCmd AT 486 : BOOL := false;
    manufacturing/mixture/cleaningValve/cmdOfValve/faults1/openCmd AT 485 : BOOL := false;
    manufacturing/mixture/cleaningValve/cmdOfValve/faults1/closedSensorFB AT 428 : BOOL := false;
    manufacturing/mixture/cleaningValve/cmdOfValve/faults1/openedSensorFB AT 429 : BOOL := false;
    manufacturing/mixture/cleaningValve/cmdOfValve/faults1/acknowledgePB AT 12 : BOOL := false;
    manufacturing/mixture/cleaningValve/cmdOfValve/faults1/generalFault AT 436 : BOOL := false;
    manufacturing/mixture/cleaningValve/cmdOfValve/faults1/closedSensorFault AT 490 : BOOL := false;
    manufacturing/mixture/cleaningValve/cmdOfValve/faults1/openedSensorFault AT 491 : BOOL := false;
    manufacturing/mixture/cleaningValve/cmdOfValve/faults1/discordanceFault AT 492 : BOOL := false;
    manufacturing/mixture/cleaningValve/cmdOfValve/faults1/presetMvt AT 861 : TIME := T#0h0m4s0ms;
    manufacturing/mixture/cleaningValve/cmdOfValve/faults1/presetDiscordance AT 865 : TIME := T#0h0m0s200ms;
    manufacturing/mixture/cleaningValve/valve/voltage380 AT 482 : BOOL := true;
    manufacturing/mixture/cleaningValve/valve/cmdSupply AT 481 : BOOL := true;
    manufacturing/mixture/cleaningValve/valve/sensorSupply AT 480 : BOOL := true;
    manufacturing/mixture/cleaningValve/valve/openCmd AT 485 : BOOL := false;
    manufacturing/mixture/cleaningValve/valve/closeCmd AT 486 : BOOL := false;
    manufacturing/mixture/cleaningValve/valve/inputFlow AT 165 : REAL := 0.0;
    manufacturing/mixture/cleaningValve/valve/openedSensor AT 429 : BOOL := false;
    manufacturing/mixture/cleaningValve/valve/closedSensor AT 428 : BOOL := false;
    manufacturing/mixture/cleaningValve/valve/outputFlow AT 164 : REAL := 0.0;
    manufacturing/mixture/cleaningValve/valve/percentOpening AT 163 : REAL := 0.0;
    manufacturing/mixture/cleaningValve/valve/increment AT 188 : REAL := 0.0;
    manufacturing/mixture/cleaningValve/valve/memoOpen AT 502 : BOOL := false;
    manufacturing/mixture/cleaningValve/valve/memoClose AT 503 : BOOL := false;
    manufacturing/mixture/cleaningValve/valve/openState AT 504 : BOOL := false;
    manufacturing/mixture/cleaningValve/valve/closeState AT 505 : BOOL := false;
    manufacturing/mixture/cleaningValve/valve/openingVal AT 189 : REAL := 0.0;
    manufacturing/mixture/cleaningValve/valve/unit AT 190 : REAL := 0.0;
    manufacturing/mixture/cleaningValve/valve/openingTime AT 191 : REAL := 2.0;
    manufacturing/mixture/cleaningValve/valve/openedSensorLogic AT 506 : BOOL := true;
    manufacturing/mixture/cleaningValve/valve/closedSensorLogic AT 507 : BOOL := true;
    manufacturing/mixture/cleaningValve/valve/flowMax AT 192 : REAL := 10000.0;
    manufacturing/mixture/cleaningValve/valve/flowPerHour AT 508 : BOOL := true;
    manufacturing/mixture/cleaningValve/valve/flowPerMinute AT 509 : BOOL := false;
    manufacturing/mixture/cleaningValve/valve/d_locking AT 510 : BOOL := false;
    manufacturing/mixture/cleaningValve/valve/v_d_locking AT 193 : REAL := 2.0;
    manufacturing/mixture/cleaningValve/valve/d_flow AT 511 : BOOL := false;
    manufacturing/mixture/cleaningValve/valve/v_d_flow AT 194 : REAL := 2.0;
    manufacturing/mixture/cleaningValve/valve/d_electrical AT 512 : BOOL := false;
    manufacturing/mixture/cleaningValve/valve/v_d_electrical AT 513 : BOOL := false;
    manufacturing/mixture/cleaningValve/valve/d_closedSensor AT 514 : BOOL := false;
    manufacturing/mixture/cleaningValve/valve/v_d_closedSensor AT 515 : BOOL := false;
    manufacturing/mixture/cleaningValve/valve/d_openedSensor AT 516 : BOOL := false;
    manufacturing/mixture/cleaningValve/valve/v_d_openedSensor AT 517 : BOOL := false;
    manufacturing/mixture/mixtureExtractingValve/acknowledgePB AT 12 : BOOL := false;
    manufacturing/mixture/mixtureExtractingValve/autoMode AT 23 : BOOL := false;
    manufacturing/mixture/mixtureExtractingValve/manualMode AT 24 : BOOL := false;
    manufacturing/mixture/mixtureExtractingValve/autoCloseCmd AT 433 : BOOL := false;
    manufacturing/mixture/mixtureExtractingValve/autoOpenCmd AT 434 : BOOL := false;
    manufacturing/mixture/mixtureExtractingValve/inputFlow AT 170 : REAL := 0.0;
    manufacturing/mixture/mixtureExtractingValve/openedSensor AT 427 : BOOL := false;
    manufacturing/mixture/mixtureExtractingValve/closedSensor AT 426 : BOOL := false;
    manufacturing/mixture/mixtureExtractingValve/generalFault AT 437 : BOOL := false;
    manufacturing/mixture/mixtureExtractingValve/outputFlow AT 172 : REAL := 0.0;
    manufacturing/mixture/mixtureExtractingValve/percentOpening AT 162 : REAL := 0.0;
    manufacturing/mixture/mixtureExtractingValve/panel1/closeValvePB AT 521 : BOOL := false;
    manufacturing/mixture/mixtureExtractingValve/panel1/openValvePB AT 522 : BOOL := false;
    manufacturing/mixture/mixtureExtractingValve/panel1/switch/leftVariable AT 521 : BOOL := false;
    manufacturing/mixture/mixtureExtractingValve/panel1/switch/rightVariable AT 522 : BOOL := false;
    manufacturing/mixture/mixtureExtractingValve/panel1/switch/leftPosition AT 525 : BOOL := false;
    manufacturing/mixture/mixtureExtractingValve/panel1/switch/middlePosition AT 526 : BOOL := false;
    manufacturing/mixture/mixtureExtractingValve/panel1/switch/rightPosition AT 527 : BOOL := false;
    manufacturing/mixture/mixtureExtractingValve/cmdOfValve/autoMode AT 23 : BOOL := false;
    manufacturing/mixture/mixtureExtractingValve/cmdOfValve/manualMode AT 24 : BOOL := false;
    manufacturing/mixture/mixtureExtractingValve/cmdOfValve/closedSensorFB AT 426 : BOOL := false;
    manufacturing/mixture/mixtureExtractingValve/cmdOfValve/openedSensorFB AT 427 : BOOL := false;
    manufacturing/mixture/mixtureExtractingValve/cmdOfValve/autoCloseCmd AT 433 : BOOL := false;
    manufacturing/mixture/mixtureExtractingValve/cmdOfValve/autoOpenCmd AT 434 : BOOL := false;
    manufacturing/mixture/mixtureExtractingValve/cmdOfValve/closeValvePB AT 521 : BOOL := false;
    manufacturing/mixture/mixtureExtractingValve/cmdOfValve/openValvePB AT 522 : BOOL := false;
    manufacturing/mixture/mixtureExtractingValve/cmdOfValve/acknowledgePB AT 12 : BOOL := false;
    manufacturing/mixture/mixtureExtractingValve/cmdOfValve/closeCmd AT 524 : BOOL := false;
    manufacturing/mixture/mixtureExtractingValve/cmdOfValve/openCmd AT 523 : BOOL := false;
    manufacturing/mixture/mixtureExtractingValve/cmdOfValve/generalFault AT 437 : BOOL := false;
    manufacturing/mixture/mixtureExtractingValve/cmdOfValve/actions/autoMode AT 23 : BOOL := false;
    manufacturing/mixture/mixtureExtractingValve/cmdOfValve/actions/manualMode AT 24 : BOOL := false;
    manufacturing/mixture/mixtureExtractingValve/cmdOfValve/actions/autoCloseCmd AT 433 : BOOL := false;
    manufacturing/mixture/mixtureExtractingValve/cmdOfValve/actions/autoOpenCmd AT 434 : BOOL := false;
    manufacturing/mixture/mixtureExtractingValve/cmdOfValve/actions/closedSensorFB AT 426 : BOOL := false;
    manufacturing/mixture/mixtureExtractingValve/cmdOfValve/actions/openedSensorFB AT 427 : BOOL := false;
    manufacturing/mixture/mixtureExtractingValve/cmdOfValve/actions/closeValvePB AT 521 : BOOL := false;
    manufacturing/mixture/mixtureExtractingValve/cmdOfValve/actions/openValvePB AT 522 : BOOL := false;
    manufacturing/mixture/mixtureExtractingValve/cmdOfValve/actions/generalFault AT 437 : BOOL := false;
    manufacturing/mixture/mixtureExtractingValve/cmdOfValve/actions/closeCmd AT 524 : BOOL := false;
    manufacturing/mixture/mixtureExtractingValve/cmdOfValve/actions/openCmd AT 523 : BOOL := false;
    manufacturing/mixture/mixtureExtractingValve/cmdOfValve/faults1/closeCmd AT 524 : BOOL := false;
    manufacturing/mixture/mixtureExtractingValve/cmdOfValve/faults1/openCmd AT 523 : BOOL := false;
    manufacturing/mixture/mixtureExtractingValve/cmdOfValve/faults1/closedSensorFB AT 426 : BOOL := false;
    manufacturing/mixture/mixtureExtractingValve/cmdOfValve/faults1/openedSensorFB AT 427 : BOOL := false;
    manufacturing/mixture/mixtureExtractingValve/cmdOfValve/faults1/acknowledgePB AT 12 : BOOL := false;
    manufacturing/mixture/mixtureExtractingValve/cmdOfValve/faults1/generalFault AT 437 : BOOL := false;
    manufacturing/mixture/mixtureExtractingValve/cmdOfValve/faults1/closedSensorFault AT 528 : BOOL := false;
    manufacturing/mixture/mixtureExtractingValve/cmdOfValve/faults1/openedSensorFault AT 529 : BOOL := false;
    manufacturing/mixture/mixtureExtractingValve/cmdOfValve/faults1/discordanceFault AT 530 : BOOL := false;
    manufacturing/mixture/mixtureExtractingValve/cmdOfValve/faults1/presetMvt AT 902 : TIME := T#0h0m4s0ms;
    manufacturing/mixture/mixtureExtractingValve/cmdOfValve/faults1/presetDiscordance AT 906 : TIME := T#0h0m0s200ms;
    manufacturing/mixture/mixtureExtractingValve/valve/voltage380 AT 520 : BOOL := true;
    manufacturing/mixture/mixtureExtractingValve/valve/cmdSupply AT 519 : BOOL := true;
    manufacturing/mixture/mixtureExtractingValve/valve/sensorSupply AT 518 : BOOL := true;
    manufacturing/mixture/mixtureExtractingValve/valve/openCmd AT 523 : BOOL := false;
    manufacturing/mixture/mixtureExtractingValve/valve/closeCmd AT 524 : BOOL := false;
    manufacturing/mixture/mixtureExtractingValve/valve/inputFlow AT 170 : REAL := 0.0;
    manufacturing/mixture/mixtureExtractingValve/valve/openedSensor AT 427 : BOOL := false;
    manufacturing/mixture/mixtureExtractingValve/valve/closedSensor AT 426 : BOOL := false;
    manufacturing/mixture/mixtureExtractingValve/valve/outputFlow AT 172 : REAL := 0.0;
    manufacturing/mixture/mixtureExtractingValve/valve/percentOpening AT 162 : REAL := 0.0;
    manufacturing/mixture/mixtureExtractingValve/valve/increment AT 198 : REAL := 0.0;
    manufacturing/mixture/mixtureExtractingValve/valve/memoOpen AT 540 : BOOL := false;
    manufacturing/mixture/mixtureExtractingValve/valve/memoClose AT 541 : BOOL := false;
    manufacturing/mixture/mixtureExtractingValve/valve/openState AT 542 : BOOL := false;
    manufacturing/mixture/mixtureExtractingValve/valve/closeState AT 543 : BOOL := false;
    manufacturing/mixture/mixtureExtractingValve/valve/openingVal AT 199 : REAL := 0.0;
    manufacturing/mixture/mixtureExtractingValve/valve/unit AT 200 : REAL := 0.0;
    manufacturing/mixture/mixtureExtractingValve/valve/openingTime AT 201 : REAL := 2.0;
    manufacturing/mixture/mixtureExtractingValve/valve/openedSensorLogic AT 544 : BOOL := true;
    manufacturing/mixture/mixtureExtractingValve/valve/closedSensorLogic AT 545 : BOOL := true;
    manufacturing/mixture/mixtureExtractingValve/valve/flowMax AT 202 : REAL := 10000.0;
    manufacturing/mixture/mixtureExtractingValve/valve/flowPerHour AT 546 : BOOL := true;
    manufacturing/mixture/mixtureExtractingValve/valve/flowPerMinute AT 547 : BOOL := false;
    manufacturing/mixture/mixtureExtractingValve/valve/d_locking AT 548 : BOOL := false;
    manufacturing/mixture/mixtureExtractingValve/valve/v_d_locking AT 203 : REAL := 2.0;
    manufacturing/mixture/mixtureExtractingValve/valve/d_flow AT 549 : BOOL := false;
    manufacturing/mixture/mixtureExtractingValve/valve/v_d_flow AT 204 : REAL := 2.0;
    manufacturing/mixture/mixtureExtractingValve/valve/d_electrical AT 550 : BOOL := false;
    manufacturing/mixture/mixtureExtractingValve/valve/v_d_electrical AT 551 : BOOL := false;
    manufacturing/mixture/mixtureExtractingValve/valve/d_closedSensor AT 552 : BOOL := false;
    manufacturing/mixture/mixtureExtractingValve/valve/v_d_closedSensor AT 553 : BOOL := false;
    manufacturing/mixture/mixtureExtractingValve/valve/d_openedSensor AT 554 : BOOL := false;
    manufacturing/mixture/mixtureExtractingValve/valve/v_d_openedSensor AT 555 : BOOL := false;
    manufacturing/mixture/mixtureWeighing/inletFlow AT 171 : REAL := 0.0;
    manufacturing/mixture/mixtureWeighing/outletFlow AT 172 : REAL := 0.0;
    manufacturing/mixture/mixtureWeighing/tankLevel AT 169 : REAL := 0.0;
    manufacturing/mixture/mixtureWeighing/percent AT 205 : REAL := 0.0;
    manufacturing/mixture/mixtureWeighing/capacity AT 206 : REAL := 600.0;
    manufacturing/mixture/mixtureWeighing/d_level AT 556 : BOOL := false;
    manufacturing/mixture/mixtureWeighing/v_d_level AT 207 : REAL := 0.0;
    manufacturing/mixture/faults1/generalFault1 AT 435 : BOOL := false;
    manufacturing/mixture/faults1/generalFault2 AT 436 : BOOL := false;
    manufacturing/mixture/faults1/generalFault3 AT 437 : BOOL := false;
    manufacturing/mixture/faults1/fault AT 52 : BOOL := false;
    manufacturing/mixture/level/measure AT 169 : REAL := 0.0;
    manufacturing/mixture/level/sensorSupply AT 425 : BOOL := true;
    manufacturing/mixture/level/realValue AT 173 : REAL := 0.0;
    manufacturing/mixture/level/intValue AT 161 : REAL := 0.0;
    manufacturing/mixture/level/dintValue AT 160 : REAL := 0.0;
    manufacturing/mixture/level/tmp AT 934 : DINT := 0;
    manufacturing/mixture/level/localValue AT 208 : REAL := 0.0;
    manufacturing/mixture/level/nbDigit AT 935 : SINT := 2;
    manufacturing/mixture/level/d_value AT 557 : BOOL := false;
    manufacturing/mixture/level/v_d_value AT 209 : REAL := 0.0;
    manufacturing/mixture/scale/inputValue AT 173 : REAL := 0.0;
    manufacturing/mixture/scale/realValue AT 159 : REAL := 0.0;
    manufacturing/mixture/scale/dintValue AT 835 : DINT := 0;
    manufacturing/mixture/scale/intValue AT 834 : INT := 0;
    manufacturing/mixture/scale/a AT 210 : REAL := 0.0;
    manufacturing/mixture/scale/b AT 211 : REAL := 0.0;
    manufacturing/mixture/scale/k AT 212 : REAL := 0.0;
    manufacturing/mixture/scale/minInput AT 213 : REAL := 0.0;
    manufacturing/mixture/scale/maxInput AT 214 : REAL := 600.0;
    manufacturing/mixture/scale/minOutput AT 215 : REAL := 0.0;
    manufacturing/mixture/scale/maxOutput AT 216 : REAL := 600.0;
    manufacturing/mixture/scale/d_scale AT 558 : BOOL := false;
    manufacturing/mixture/scale/v_d_scale AT 217 : REAL := 0.0;
    manufacturing/faults1/fault3 AT 52 : BOOL := false;
    manufacturing/faults1/fault2 AT 53 : BOOL := false;
    manufacturing/faults1/fault1 AT 54 : BOOL := false;
    manufacturing/faults1/generalFault AT 14 : BOOL := false;
  END_VAR
END_CONFIGURATION
